  MoveL 8481 to (467.23, 529.71, 152) mm, rotated rx -180 ry 0 rz 160 deg; joints [10.696, 50.173, 8.575, -145.223, 63.505, 162.787]
  Set speed (16.9 mm/s)
  Call Extruder(111.55322)
  MoveL 8482 to (466.64, 529.05, 152) mm, rotated rx -180 ry 0 rz 160 deg; joints [10.622, 50.069, 8.779, -145.33, 63.566, 162.886]
  Set speed (16.9 mm/s)
  Call Extruder(114.56277)
  MoveL 8483 to (466.06, 528.36, 152) mm, rotated rx 180 ry 0 rz 160 deg; joints [10.545, 49.965, 8.983, -145.44, 63.625, 162.986]
  Call Extruder(117.70590)
  MoveL 8484 to (465.46, 527.63, 152) mm, rotated rx -180 ry 0 rz 160 deg; joints [10.463, 49.858, 9.191, -145.557, 63.685, 163.089]
  Set speed (16.9 mm/s)
  Call Extruder(120.63235)
  MoveL 8485 to (464.92, 526.94, 152) mm, rotated rx -180 ry 0 rz 160 deg; joints [10.384, 49.761, 9.381, -145.667, 63.739, 163.185]
  Call Extruder(123.51753)
  MoveL 8486 to (464.4, 526.25, 152) mm, rotated rx -180 ry 0 rz 160 deg; joints [10.304, 49.667, 9.565, -145.777, 63.79, 163.279]
  Set speed (16.9 mm/s)
  Call Extruder(126.65561)
  MoveL 8487 to (463.85, 525.49, 152) mm, rotated rx 180 ry 0 rz 160 deg; joints [10.215, 49.568, 9.76, -145.898, 63.844, 163.381]
  Set speed (16.9 mm/s)
  Call Extruder(130.52968)
  MoveL 8488 to (463.19, 524.53, 152) mm, rotated rx 180 ry 0 rz 160 deg; joints [10.102, 49.448, 9.995, -146.05, 63.907, 163.505]
  Call Extruder(135.63472)
  MoveL 8489 to (462.37, 523.24, 152) mm, rotated rx 180 ry 0 rz 160 deg; joints [9.948, 49.296, 10.292, -146.255, 63.984, 163.668]
  Set speed (16.9 mm/s)
  Call Extruder(138.64613)
  MoveL 8490 to (461.9, 522.47, 152) mm, rotated rx 180 ry 0 rz 160 deg; joints [9.855, 49.21, 10.461, -146.377, 64.027, 163.763]
  Set speed (16.9 mm/s)
  Call Extruder(141.85812)
  MoveL 8491 to (461.42, 521.64, 152) mm, rotated rx 180 ry 0 rz 160 deg; joints [9.753, 49.12, 10.637, -146.509, 64.07, 163.864]
  Set speed (16.9 mm/s)
  Call Extruder(144.69950)
  MoveL 8492 to (461.01, 520.89, 152) mm, rotated rx 180 ry 0 rz 160 deg; joints [9.661, 49.043, 10.788, -146.627, 64.107, 163.952]
  Set speed (16.9 mm/s)
  Call Extruder(147.76672)
  MoveL 8493 to (460.58, 520.07, 152) mm, rotated rx -180 ry 0 rz 160 deg; joints [9.56, 48.962, 10.946, -146.755, 64.144, 164.046]
  Set speed (16.9 mm/s)
  Call Extruder(150.71748)
  MoveL 8494 to (460.19, 519.28, 152) mm, rotated rx 180 ry 0 rz 160 deg; joints [9.461, 48.887, 11.094, -146.88, 64.177, 164.136]
  Call Extruder(156.72530)
  MoveL 8495 to (459.44, 517.64, 152) mm, rotated rx 180 ry 0 rz 160 deg; joints [9.255, 48.741, 11.38, -147.137, 64.239, 164.317]
  Call Extruder(162.74277)
  MoveL 8496 to (458.75, 515.98, 152) mm, rotated rx 180 ry 0 rz 160 deg; joints [9.042, 48.605, 11.647, -147.399, 64.292, 164.494]
  Set speed (16.9 mm/s)
  Call Extruder(164.64160)
  MoveL 8497 to (458.55, 515.44, 152) mm, rotated rx -180 ry 0 rz 160 deg; joints [8.974, 48.564, 11.727, -147.483, 64.306, 164.549]
  Set speed (16.9 mm/s)
  Call Extruder(168.87909)
  MoveL 8498 to (458.12, 514.25, 152) mm, rotated rx 180 ry 0 rz 160 deg; joints [8.819, 48.477, 11.898, -147.67, 64.336, 164.671]
  Set speed (16.9 mm/s)
  Call Extruder(174.83651)
  MoveL 8499 to (457.58, 512.55, 152) mm, rotated rx 180 ry 0 rz 160 deg; joints [8.596, 48.363, 12.122, -147.936, 64.37, 164.839]
  Call Extruder(180.93408)
  MoveL 8500 to (457.1, 510.79, 152) mm, rotated rx 180 ry 0 rz 160 deg; joints [8.363, 48.257, 12.33, -148.211, 64.396, 165.007]
  Set speed (16.9 mm/s)
  Call Extruder(186.95183)
  MoveL 8501 to (456.7, 509.03, 152) mm, rotated rx -180 ry 0 rz 160 deg; joints [8.128, 48.165, 12.512, -148.485, 64.412, 165.167]
  Set speed (16.9 mm/s)
  Call Extruder(193.18882)
  MoveL 8502 to (456.36, 507.19, 152) mm, rotated rx 180 ry 0 rz 160 deg; joints [7.881, 48.079, 12.679, -148.772, 64.419, 165.33]
  Set speed (16.9 mm/s)
  Call Extruder(199.22762)
  MoveL 8503 to (456.1, 505.4, 152) mm, rotated rx 180 ry 0 rz 160 deg; joints [7.637, 48.008, 12.818, -149.05, 64.416, 165.482]
  Set speed (16.9 mm/s)
  Call Extruder(205.26140)
  MoveL 8504 to (455.91, 503.6, 152) mm, rotated rx -180 ry 0 rz 160 deg; joints [7.39, 47.949, 12.936, -149.329, 64.404, 165.629]
  Set speed (16.9 mm/s)
  Call Extruder(211.19905)
  MoveL 8505 to (455.8, 501.82, 152) mm, rotated rx -180 ry 0 rz 160 deg; joints [7.145, 47.901, 13.029, -149.603, 64.382, 165.768]
  Set speed (16.9 mm/s)
  Call Extruder(217.23836)
  MoveL 8506 to (455.76, 500.01, 152) mm, rotated rx -180 ry 0 rz 160 deg; joints [6.894, 47.864, 13.102, -149.883, 64.352, 165.905]
  Set speed (16.9 mm/s)
  Call Extruder(222.75136)
  MoveL 8507 to (455.8, 498.36, 152) mm, rotated rx -180 ry 0 rz 160 deg; joints [6.662, 47.841, 13.147, -150.137, 64.315, 166.025]
  Set speed (16.9 mm/s)
  Call Extruder(228.09484)
  MoveL 8508 to (455.89, 496.76, 152) mm, rotated rx -180 ry 0 rz 160 deg; joints [6.438, 47.828, 13.173, -150.382, 64.272, 166.137]
  Call Extruder(233.51834)
  MoveL 8509 to (456.03, 495.14, 152) mm, rotated rx -180 ry 0 rz 160 deg; joints [6.209, 47.823, 13.182, -150.629, 64.222, 166.247]
  Call Extruder(238.82118)
  MoveL 8510 to (456.24, 493.56, 152) mm, rotated rx -180 ry 0 rz 160 deg; joints [5.986, 47.828, 13.172, -150.869, 64.164, 166.349]
  Set speed (16.9 mm/s)
  Call Extruder(244.49040)
  MoveL 8511 to (456.52, 491.89, 152) mm, rotated rx 180 ry 0 rz 160 deg; joints [5.748, 47.843, 13.142, -151.123, 64.096, 166.453]
  Call Extruder(249.82084)
  MoveL 8512 to (456.84, 490.32, 152) mm, rotated rx -180 ry 0 rz 160 deg; joints [5.525, 47.867, 13.096, -151.359, 64.024, 166.547]
  Set speed (16.9 mm/s)
  Call Extruder(255.25540)
  MoveL 8513 to (457.22, 488.74, 152) mm, rotated rx 180 ry 0 rz 160 deg; joints [5.298, 47.9, 13.03, -151.596, 63.943, 166.637]
  Set speed (16.9 mm/s)
  Call Extruder(260.70317)
  MoveL 8514 to (457.67, 487.17, 152) mm, rotated rx 180 ry 0 rz 160 deg; joints [5.073, 47.943, 12.946, -151.83, 63.855, 166.723]
  Set speed (16.9 mm/s)
  Call Extruder(266.12310)
  MoveL 8515 to (458.17, 485.63, 152) mm, rotated rx -180 ry 0 rz 160 deg; joints [4.851, 47.995, 12.844, -152.06, 63.76, 166.803]
  Set speed (16.9 mm/s)
  Call Extruder(271.65144)
  MoveL 8516 to (458.73, 484.07, 152) mm, rotated rx 180 ry 0 rz 160 deg; joints [4.628, 48.057, 12.722, -152.289, 63.656, 166.879]
  Call Extruder(277.08602)
  MoveL 8517 to (459.35, 482.56, 152) mm, rotated rx -180 ry 0 rz 160 deg; joints [4.411, 48.128, 12.584, -152.509, 63.546, 166.949]
  Call Extruder(282.51502)
  MoveL 8518 to (460.02, 481.08, 152) mm, rotated rx 180 ry 0 rz 160 deg; joints [4.197, 48.207, 12.428, -152.724, 63.43, 167.013]
  Call Extruder(287.86511)
  MoveL 8519 to (460.73, 479.64, 152) mm, rotated rx 180 ry 0 rz 160 deg; joints [3.99, 48.294, 12.257, -152.931, 63.309, 167.072]
  Set speed (16.9 mm/s)
  Call Extruder(293.30641)
  MoveL 8520 to (461.51, 478.21, 152) mm, rotated rx 180 ry 0 rz 160 deg; joints [3.783, 48.391, 12.066, -153.135, 63.18, 167.126]
  Set speed (16.9 mm/s)
  Call Extruder(298.82528)
  MoveL 8521 to (462.35, 476.78, 152) mm, rotated rx 180 ry 0 rz 160 deg; joints [3.578, 48.499, 11.854, -153.335, 63.041, 167.175]
  Set speed (16.9 mm/s)
  Call Extruder(304.15599)
  MoveL 8522 to (463.21, 475.44, 152) mm, rotated rx -180 ry 0 rz 160 deg; joints [3.385, 48.612, 11.634, -153.523, 62.902, 167.217]
  Set speed (16.9 mm/s)
  Call Extruder(309.59991)
  MoveL 8523 to (464.15, 474.1, 152) mm, rotated rx 180 ry 0 rz 160 deg; joints [3.192, 48.735, 11.392, -153.707, 62.753, 167.254]
  Set speed (16.9 mm/s)
  Call Extruder(315.02617)
  MoveL 8524 to (465.12, 472.8, 152) mm, rotated rx -180 ry 0 rz 160 deg; joints [3.005, 48.866, 11.136, -153.883, 62.599, 167.286]
  Set speed (16.9 mm/s)
  Call Extruder(320.54632)
  MoveL 8525 to (466.16, 471.51, 152) mm, rotated rx 180 ry 0 rz 160 deg; joints [2.821, 49.008, 10.858, -154.055, 62.436, 167.312]
  Set speed (16.9 mm/s)
  Call Extruder(325.88657)
  MoveL 8526 to (467.22, 470.31, 152) mm, rotated rx 180 ry 0 rz 160 deg; joints [2.648, 49.152, 10.574, -154.213, 62.273, 167.332]
  Call Extruder(331.41574)
  MoveL 8527 to (468.35, 469.1, 152) mm, rotated rx -180 ry 0 rz 160 deg; joints [2.476, 49.31, 10.265, -154.369, 62.099, 167.346]
  Set speed (16.9 mm/s)
  Call Extruder(336.75261)
  MoveL 8528 to (469.49, 467.97, 152) mm, rotated rx -180 ry 0 rz 160 deg; joints [2.315, 49.47, 9.952, -154.511, 61.926, 167.355]
  Set speed (16.9 mm/s)
  Call Extruder(342.18977)
  MoveL 8529 to (470.69, 466.87, 152) mm, rotated rx 180 ry 0 rz 160 deg; joints [2.159, 49.64, 9.619, -154.647, 61.744, 167.357]
  Call Extruder(347.70524)
  MoveL 8530 to (471.95, 465.8, 152) mm, rotated rx 180 ry 0 rz 160 deg; joints [2.006, 49.819, 9.268, -154.776, 61.555, 167.354]
  Set speed (16.9 mm/s)
  Call Extruder(353.50911)
  MoveL 8531 to (473.32, 464.72, 152) mm, rotated rx 180 ry 0 rz 160 deg; joints [1.854, 50.016, 8.883, -154.902, 61.352, 167.343]
  Set speed (16.9 mm/s)
  Call Extruder(357.99277)
  MoveL 8532 to (474.4, 463.93, 152) mm, rotated rx -180 ry 0 rz 160 deg; joints [1.742, 50.172, 8.576, -154.991, 61.191, 167.331]
  Set speed (16.9 mm/s)
  Call Extruder(363.92441)
  MoveL 8533 to (475.87, 462.93, 152) mm, rotated rx -180 ry 0 rz 160 deg; joints [1.602, 50.387, 8.156, -155.1, 60.974, 167.307]
  Set speed (16.9 mm/s)
  Call Extruder(369.45306)
  MoveL 8534 to (477.27, 462.05, 152) mm, rotated rx -180 ry 0 rz 160 deg; joints [1.479, 50.593, 7.752, -155.191, 60.768, 167.279]
  Set speed (16.9 mm/s)
  Call Extruder(374.88475)
  MoveL 8535 to (478.68, 461.24, 152) mm, rotated rx -180 ry 0 rz 160 deg; joints [1.365, 50.803, 7.343, -155.271, 60.561, 167.245]
  Call Extruder(380.22948)
  MoveL 8536 to (480.1, 460.5, 152) mm, rotated rx -180 ry 0 rz 160 deg; joints [1.261, 51.014, 6.93, -155.34, 60.355, 167.206]
  Call Extruder(385.74670)
  MoveL 8537 to (481.59, 459.78, 152) mm, rotated rx -180 ry 0 rz 160 deg; joints [1.162, 51.237, 6.493, -155.401, 60.138, 167.159]
  Set speed (16.9 mm/s)
  Call Extruder(391.17918)
  MoveL 8538 to (483.09, 459.13, 152) mm, rotated rx 180 ry 0 rz 160 deg; joints [1.072, 51.463, 6.052, -155.451, 59.922, 167.106]
  Call Extruder(396.52455)
  MoveL 8539 to (484.58, 458.54, 152) mm, rotated rx -180 ry 0 rz 160 deg; joints [0.99, 51.689, 5.609, -155.49, 59.708, 167.048]
  Set speed (16.9 mm/s)
  Call Extruder(402.01351)
  MoveL 8540 to (486.13, 458, 152) mm, rotated rx 180 ry 0 rz 160 deg; joints [0.915, 51.926, 5.146, -155.52, 59.485, 166.982]
  Call Extruder(407.42300)
  MoveL 8541 to (487.68, 457.52, 152) mm, rotated rx 180 ry 0 rz 160 deg; joints [0.849, 52.164, 4.681, -155.539, 59.264, 166.911]
  Set speed (16.9 mm/s)
  Call Extruder(412.57446)
  MoveL 8542 to (489.17, 457.11, 152) mm, rotated rx -180 ry 0 rz 160 deg; joints [0.793, 52.395, 4.231, -155.548, 59.051, 166.838]
  Set speed (16.9 mm/s)
  Call Extruder(418.05427)
  MoveL 8543 to (490.77, 456.74, 152) mm, rotated rx 180 ry 0 rz 160 deg; joints [0.742, 52.643, 3.746, -155.547, 58.824, 166.754]
  Call Extruder(423.53685)
  MoveL 8544 to (492.38, 456.43, 152) mm, rotated rx -180 ry 0 rz 160 deg; joints [0.699, 52.896, 3.253, -155.536, 58.595, 166.663]
  Set speed (16.9 mm/s)
  Call Extruder(429.18834)
  MoveL 8545 to (494.06, 456.17, 152) mm, rotated rx 180 ry 0 rz 160 deg; joints [0.662, 53.159, 2.739, -155.514, 58.359, 166.563]
  Set speed (16.9 mm/s)
  Call Extruder(434.59269)
  MoveL 8546 to (495.66, 455.98, 152) mm, rotated rx -180 ry 0 rz 160 deg; joints [0.636, 53.414, 2.242, -155.482, 58.132, 166.461]
  Set speed (16.9 mm/s)
  Call Extruder(440.01240)
  MoveL 8547 to (497.28, 455.85, 152) mm, rotated rx 180 ry 0 rz 160 deg; joints [0.617, 53.672, 1.739, -155.44, 57.905, 166.352]
  Set speed (16.9 mm/s)
  Call Extruder(445.51598)
  MoveL 8548 to (498.93, 455.78, 152) mm, rotated rx -180 ry 0 rz 160 deg; joints [0.606, 53.936, 1.224, -155.388, 57.674, 166.236]
  Set speed (16.9 mm/s)
  Call Extruder(450.85230)
  MoveL 8549 to (500.53, 455.77, 152) mm, rotated rx 180 ry 0 rz 160 deg; joints [0.602, 54.194, 0.722, -155.327, 57.451, 166.117]
  Set speed (16.9 mm/s)
  Call Extruder(456.35038)
  MoveL 8550 to (502.18, 455.82, 152) mm, rotated rx -180 ry 0 rz 160 deg; joints [0.606, 54.462, 0.2, -155.254, 57.222, 165.988]
  Set speed (16.9 mm/s)
  Call Extruder(461.73242)
  MoveL 8551 to (503.79, 455.93, 152) mm, rotated rx -180 ry 0 rz 160 deg; joints [0.618, 54.725, -0.312, -155.173, 56.998, 165.857]
  Set speed (16.9 mm/s)
  Call Extruder(467.24230)
  MoveL 8552 to (505.43, 456.1, 152) mm, rotated rx 180 ry 0 rz 160 deg; joints [0.637, 54.995, -0.838, -155.08, 56.771, 165.716]
  Set speed (16.9 mm/s)
  Call Extruder(472.59761)
  MoveL 8553 to (507.02, 456.33, 152) mm, rotated rx 180 ry 0 rz 160 deg; joints [0.664, 55.258, -1.349, -154.981, 56.552, 165.574]
  Call Extruder(478.00070)
  MoveL 8554 to (508.62, 456.61, 152) mm, rotated rx 180 ry 0 rz 160 deg; joints [0.697, 55.523, -1.866, -154.871, 56.333, 165.424]
  Set speed (16.9 mm/s)
  Call Extruder(482.76006)
  MoveL 8555 to (510.01, 456.91, 152) mm, rotated rx -180 ry 0 rz 160 deg; joints [0.732, 55.757, -2.32, -154.767, 56.142, 165.289]
  Call Extruder(488.88102)
  MoveL 8556 to (511.79, 457.37, 152) mm, rotated rx -180 ry 0 rz 160 deg; joints [0.786, 56.057, -2.904, -154.624, 55.899, 165.108]
  Set speed (16.9 mm/s)
  Call Extruder(494.30171)
  MoveL 8557 to (513.34, 457.83, 152) mm, rotated rx 180 ry 0 rz 160 deg; joints [0.84, 56.322, -3.419, -154.487, 55.687, 164.942]
  Call Extruder(499.82708)
  MoveL 8558 to (514.91, 458.36, 152) mm, rotated rx 180 ry 0 rz 160 deg; joints [0.903, 56.59, -3.942, -154.339, 55.475, 164.768]
  Call Extruder(505.16704)
  MoveL 8559 to (516.41, 458.93, 152) mm, rotated rx 180 ry 0 rz 160 deg; joints [0.97, 56.849, -4.444, -154.187, 55.273, 164.595]
  Set speed (16.9 mm/s)
  Call Extruder(510.69488)
  MoveL 8560 to (517.94, 459.57, 152) mm, rotated rx -180 ry 0 rz 160 deg; joints [1.045, 57.114, -4.96, -154.022, 55.068, 164.411]
  Set speed (16.9 mm/s)
  Call Extruder(516.02911)
  MoveL 8561 to (519.39, 460.24, 152) mm, rotated rx -180 ry 0 rz 160 deg; joints [1.125, 57.368, -5.453, -153.855, 54.874, 164.229]
  Set speed (16.9 mm/s)
  Call Extruder(521.56196)
  MoveL 8562 to (520.87, 461, 152) mm, rotated rx 180 ry 0 rz 160 deg; joints [1.213, 57.629, -5.959, -153.674, 54.678, 164.036]
  Set speed (16.9 mm/s)
  Call Extruder(526.98931)
  MoveL 8563 to (522.28, 461.79, 152) mm, rotated rx 180 ry 0 rz 160 deg; joints [1.306, 57.882, -6.45, -153.49, 54.491, 163.842]
  Set speed (16.9 mm/s)
  Call Extruder(532.32683)
  MoveL 8564 to (523.65, 462.62, 152) mm, rotated rx 180 ry 0 rz 160 deg; joints [1.403, 58.127, -6.926, -153.301, 54.311, 163.649]
  Set speed (16.9 mm/s)
  Call Extruder(537.85094)
  MoveL 8565 to (525.03, 463.53, 152) mm, rotated rx -180 ry 0 rz 160 deg; joints [1.509, 58.378, -7.412, -153.1, 54.131, 163.445]
  Set speed (16.9 mm/s)
  Call Extruder(543.19366)
  MoveL 8566 to (526.34, 464.46, 152) mm, rotated rx -180 ry 0 rz 160 deg; joints [1.616, 58.616, -7.874, -152.898, 53.963, 163.244]
  Set speed (16.9 mm/s)
  Call Extruder(548.66042)
  MoveL 8567 to (527.64, 465.47, 152) mm, rotated rx 180 ry 0 rz 160 deg; joints [1.732, 58.855, -8.338, -152.686, 53.796, 163.036]
  Call Extruder(554.09541)
  MoveL 8568 to (528.89, 466.51, 152) mm, rotated rx 180 ry 0 rz 160 deg; joints [1.852, 59.088, -8.79, -152.47, 53.637, 162.827]
  Set speed (16.9 mm/s)
  Call Extruder(559.59156)
  MoveL 8569 to (530.12, 467.61, 152) mm, rotated rx -180 ry 0 rz 160 deg; joints [1.979, 59.319, -9.237, -152.246, 53.483, 162.613]
  Call Extruder(564.97166)
  MoveL 8570 to (531.28, 468.73, 152) mm, rotated rx 180 ry 0 rz 160 deg; joints [2.107, 59.539, -9.664, -152.021, 53.339, 162.401]
  Set speed (16.9 mm/s)
  Call Extruder(567.88723)
  MoveL 8571 to (531.89, 469.35, 152) mm, rotated rx -180 ry 0 rz 160 deg; joints [2.179, 59.656, -9.891, -151.898, 53.264, 162.286]
  Call Extruder(570.83929)
  MoveL 8572 to (532.5, 469.99, 152) mm, rotated rx 180 ry 0 rz 160 deg; joints [2.253, 59.773, -10.117, -151.771, 53.19, 162.169]
  Set speed (16.9 mm/s)
  Call Extruder(573.85291)
  MoveL 8573 to (533.11, 470.66, 152) mm, rotated rx -180 ry 0 rz 160 deg; joints [2.329, 59.891, -10.345, -151.641, 53.116, 162.049]
  Set speed (16.9 mm/s)
  Call Extruder(576.90040)
  MoveL 8574 to (533.7, 471.35, 152) mm, rotated rx -180 ry 0 rz 160 deg; joints [2.408, 60.007, -10.571, -151.508, 53.045, 161.928]
  Set speed (16.9 mm/s)
  Call Extruder(579.88352)
  MoveL 8575 to (534.27, 472.04, 152) mm, rotated rx 180 ry 0 rz 160 deg; joints [2.486, 60.119, -10.788, -151.377, 52.977, 161.809]
  Set speed (16.9 mm/s)
  Call Extruder(582.95706)
  MoveL 8576 to (534.85, 472.76, 152) mm, rotated rx 180 ry 0 rz 160 deg; joints [2.569, 60.233, -11.008, -151.241, 52.909, 161.686]
  Set speed (16.9 mm/s)
  Call Extruder(585.93160)
  MoveL 8577 to (535.39, 473.47, 152) mm, rotated rx 180 ry 0 rz 160 deg; joints [2.649, 60.341, -11.217, -151.108, 52.846, 161.567]
  Set speed (16.9 mm/s)
  Call Extruder(589.06730)
  MoveL 8578 to (535.95, 474.23, 152) mm, rotated rx -180 ry 0 rz 160 deg; joints [2.735, 60.452, -11.432, -150.967, 52.782, 161.442]
  Set speed (16.9 mm/s)
  Call Extruder(591.96265)
  MoveL 8579 to (536.45, 474.94, 152) mm, rotated rx -180 ry 0 rz 160 deg; joints [2.816, 60.553, -11.627, -150.836, 52.726, 161.326]
  Set speed (16.9 mm/s)
  Call Extruder(594.99815)
  MoveL 8580 to (536.95, 475.69, 152) mm, rotated rx 180 ry 0 rz 160 deg; joints [2.902, 60.656, -11.827, -150.698, 52.669, 161.205]
  Call Extruder(598.05624)
  MoveL 8581 to (537.45, 476.46, 152) mm, rotated rx -180 ry 0 rz 160 deg; joints [2.99, 60.758, -12.024, -150.558, 52.614, 161.083]
  Call Extruder(601.06718)
  MoveL 8582 to (537.92, 477.23, 152) mm, rotated rx -180 ry 0 rz 160 deg; joints [3.077, 60.855, -12.212, -150.42, 52.564, 160.963]
  Set speed (16.9 mm/s)
  Call Extruder(604.06606)
  MoveL 8583 to (538.38, 478.01, 152) mm, rotated rx -180 ry 0 rz 160 deg; joints [3.165, 60.95, -12.397, -150.281, 52.515, 160.844]
  Set speed (16.9 mm/s)
  Call Extruder(608.88178)
  MoveL 8584 to (539.08, 479.27, 152) mm, rotated rx 180 ry 0 rz 160 deg; joints [3.308, 61.098, -12.682, -150.059, 52.442, 160.654]
  Call Extruder(613.09280)
  MoveL 8585 to (539.65, 480.39, 152) mm, rotated rx 180 ry 0 rz 160 deg; joints [3.435, 61.22, -12.92, -149.863, 52.385, 160.489]
  Set speed (16.9 mm/s)
  Call Extruder(616.12747)
  MoveL 8586 to (540.04, 481.21, 152) mm, rotated rx 180 ry 0 rz 160 deg; joints [3.528, 61.306, -13.085, -149.721, 52.347, 160.371]
  Set speed (16.9 mm/s)
  Call Extruder(619.14351)
  MoveL 8587 to (540.42, 482.03, 152) mm, rotated rx 180 ry 0 rz 160 deg; joints [3.621, 61.389, -13.245, -149.58, 52.312, 160.254]
  Set speed (16.9 mm/s)
  Call Extruder(625.34531)
  MoveL 8588 to (541.14, 483.75, 152) mm, rotated rx 180 ry 0 rz 160 deg; joints [3.815, 61.549, -13.555, -149.291, 52.249, 160.016]
  Set speed (16.9 mm/s)
  Call Extruder(631.18422)
  MoveL 8589 to (541.75, 485.39, 152) mm, rotated rx -180 ry 0 rz 160 deg; joints [4.001, 61.689, -13.827, -149.018, 52.2, 159.796]
  Set speed (16.9 mm/s)
  Call Extruder(637.24238)
  MoveL 8590 to (542.31, 487.11, 152) mm, rotated rx 180 ry 0 rz 160 deg; joints [4.196, 61.824, -14.087, -148.735, 52.16, 159.571]
  Set speed (16.9 mm/s)
  Call Extruder(643.43589)
  MoveL 8591 to (542.82, 488.9, 152) mm, rotated rx 180 ry 0 rz 160 deg; joints [4.399, 61.949, -14.329, -148.448, 52.132, 159.347]
  Set speed (16.9 mm/s)
  Call Extruder(649.40759)
  MoveL 8592 to (543.23, 490.64, 152) mm, rotated rx 180 ry 0 rz 160 deg; joints [4.597, 62.057, -14.538, -148.172, 52.116, 159.136]
  Set speed (16.9 mm/s)
  Call Extruder(655.48431)
  MoveL 8593 to (543.58, 492.43, 152) mm, rotated rx 180 ry 0 rz 160 deg; joints [4.8, 62.155, -14.726, -147.894, 52.112, 158.927]
  Set speed (16.9 mm/s)
  Call Extruder(661.50732)
  MoveL 8594 to (543.85, 494.21, 152) mm, rotated rx 180 ry 0 rz 160 deg; joints [5.003, 62.239, -14.889, -147.622, 52.119, 158.727]
  Call Extruder(667.39278)
  MoveL 8595 to (544.05, 495.96, 152) mm, rotated rx -180 ry 0 rz 160 deg; joints [5.203, 62.308, -15.023, -147.359, 52.137, 158.538]
  Set speed (16.9 mm/s)
  Call Extruder(673.59529)
  MoveL 8596 to (544.18, 497.82, 152) mm, rotated rx -180 ry 0 rz 160 deg; joints [5.415, 62.369, -15.14, -147.085, 52.167, 158.346]
  Set speed (16.9 mm/s)
  Call Extruder(679.61986)
  MoveL 8597 to (544.23, 499.63, 152) mm, rotated rx 180 ry 0 rz 160 deg; joints [5.622, 62.414, -15.227, -146.824, 52.209, 158.168]
  Call Extruder(685.75246)
  MoveL 8598 to (544.21, 501.46, 152) mm, rotated rx 180 ry 0 rz 160 deg; joints [5.834, 62.446, -15.289, -146.563, 52.263, 157.995]
  Call Extruder(691.68280)
  MoveL 8599 to (544.12, 503.24, 152) mm, rotated rx 180 ry 0 rz 160 deg; joints [6.039, 62.464, -15.324, -146.315, 52.326, 157.836]
  Set speed (16.9 mm/s)
  Call Extruder(697.71345)
  MoveL 8600 to (543.95, 505.04, 152) mm, rotated rx 180 ry 0 rz 160 deg; joints [6.248, 62.469, -15.334, -146.069, 52.401, 157.684]
  Set speed (16.9 mm/s)
  Call Extruder(703.84606)
  MoveL 8601 to (543.7, 506.86, 152) mm, rotated rx 180 ry 0 rz 160 deg; joints [6.46, 62.46, -15.316, -145.825, 52.489, 157.539]
  Set speed (16.9 mm/s)
  Call Extruder(709.77348)
  MoveL 8602 to (543.39, 508.61, 152) mm, rotated rx -180 ry 0 rz 160 deg; joints [6.665, 62.438, -15.274, -145.596, 52.585, 157.408]
  Call Extruder(715.61424)
  MoveL 8603 to (543.01, 510.32, 152) mm, rotated rx 180 ry 0 rz 160 deg; joints [6.866, 62.404, -15.208, -145.376, 52.688, 157.289]
  Set speed (16.9 mm/s)
  Call Extruder(721.80459)
  MoveL 8604 to (542.54, 512.12, 152) mm, rotated rx -180 ry 0 rz 160 deg; joints [7.079, 62.354, -15.112, -145.15, 52.809, 157.173]
  Set speed (16.9 mm/s)
  Call Extruder(727.90138)
  MoveL 8605 to (542, 513.87, 152) mm, rotated rx 180 ry 0 rz 160 deg; joints [7.287, 62.292, -14.991, -144.934, 52.937, 157.07]
  Call Extruder(734.04898)
  MoveL 8606 to (541.39, 515.6, 152) mm, rotated rx 180 ry 0 rz 160 deg; joints [7.496, 62.216, -14.844, -144.725, 53.077, 156.976]
  Set speed (16.9 mm/s)
  Call Extruder(739.76790)
  MoveL 8607 to (540.75, 517.2, 152) mm, rotated rx 180 ry 0 rz 160 deg; joints [7.688, 62.132, -14.683, -144.537, 53.216, 156.9]
  Set speed (16.9 mm/s)
  Call Extruder(745.87332)
  MoveL 8608 to (540.01, 518.87, 152) mm, rotated rx 180 ry 0 rz 160 deg; joints [7.892, 62.031, -14.487, -144.345, 53.373, 156.829]
  Set speed (16.9 mm/s)
  Call Extruder(748.95640)
  MoveL 8609 to (539.61, 519.7, 152) mm, rotated rx 180 ry 0 rz 160 deg; joints [7.994, 61.975, -14.379, -144.251, 53.455, 156.797]
  Set speed (16.9 mm/s)
  Call Extruder(751.90685)
  MoveL 8610 to (539.2, 520.49, 152) mm, rotated rx -180 ry 0 rz 160 deg; joints [8.091, 61.918, -14.269, -144.162, 53.536, 156.77]
  Set speed (16.9 mm/s)
  Call Extruder(755.31926)
  MoveL 8611 to (538.72, 521.39, 152) mm, rotated rx 180 ry 0 rz 160 deg; joints [8.203, 61.85, -14.136, -144.063, 53.632, 156.741]
  Set speed (16.9 mm/s)
  Call Extruder(758.08631)
  MoveL 8612 to (538.31, 522.11, 152) mm, rotated rx 180 ry 0 rz 160 deg; joints [8.292, 61.79, -14.021, -143.984, 53.713, 156.721]
  Set speed (16.9 mm/s)
  Call Extruder(763.51652)
  MoveL 8613 to (537.48, 523.5, 152) mm, rotated rx 180 ry 0 rz 160 deg; joints [8.467, 61.668, -13.786, -143.834, 53.874, 156.686]
  Set speed (16.9 mm/s)
  Call Extruder(766.36303)
  MoveL 8614 to (537.01, 524.22, 152) mm, rotated rx 180 ry 0 rz 160 deg; joints [8.558, 61.6, -13.653, -143.759, 53.961, 156.672]
  Set speed (16.9 mm/s)
  Call Extruder(771.70559)
  MoveL 8615 to (536.11, 525.55, 152) mm, rotated rx 180 ry 0 rz 160 deg; joints [8.726, 61.466, -13.394, -143.621, 54.129, 156.651]
  Set speed (16.9 mm/s)
  Call Extruder(776.09850)
  MoveL 8616 to (535.33, 526.61, 152) mm, rotated rx 180 ry 0 rz 160 deg; joints [8.863, 61.348, -13.166, -143.514, 54.272, 156.642]
  Set speed (16.9 mm/s)
  Call Extruder(779.07385)
  MoveL 8617 to (534.79, 527.32, 152) mm, rotated rx 180 ry 0 rz 160 deg; joints [8.954, 61.265, -13.007, -143.444, 54.37, 156.638]
  Set speed (16.9 mm/s)
  Call Extruder(782.31334)
  MoveL 8618 to (534.18, 528.07, 152) mm, rotated rx 180 ry 0 rz 160 deg; joints [9.053, 61.172, -12.826, -143.369, 54.479, 156.637]
  Set speed (16.9 mm/s)
  Call Extruder(785.08810)
  MoveL 8619 to (533.65, 528.71, 152) mm, rotated rx 180 ry 0 rz 160 deg; joints [9.136, 61.09, -12.668, -143.308, 54.574, 156.639]
  Set speed (16.9 mm/s)
  Call Extruder(788.18970)
  MoveL 8620 to (533.04, 529.41, 152) mm, rotated rx 180 ry 0 rz 160 deg; joints [9.229, 60.996, -12.485, -143.241, 54.681, 156.643]
  Call Extruder(791.17742)
  MoveL 8621 to (532.44, 530.08, 152) mm, rotated rx 180 ry 0 rz 160 deg; joints [9.317, 60.903, -12.305, -143.179, 54.785, 156.649]
  Call Extruder(794.30638)
  MoveL 8622 to (531.79, 530.76, 152) mm, rotated rx 180 ry 0 rz 160 deg; joints [9.409, 60.803, -12.112, -143.116, 54.897, 156.659]
  Set speed (16.9 mm/s)
  Call Extruder(797.24483)
  MoveL 8623 to (531.17, 531.38, 152) mm, rotated rx -180 ry 0 rz 160 deg; joints [9.493, 60.706, -11.924, -143.059, 55.002, 156.671]
  Set speed (16.9 mm/s)
  Call Extruder(800.21250)
  MoveL 8624 to (530.53, 532, 152) mm, rotated rx -180 ry 0 rz 160 deg; joints [9.578, 60.606, -11.731, -143.004, 55.111, 156.685]
  Call Extruder(803.23832)
  MoveL 8625 to (529.87, 532.62, 152) mm, rotated rx 180 ry 0 rz 160 deg; joints [9.663, 60.502, -11.529, -142.949, 55.222, 156.703]
  Set speed (16.9 mm/s)
  Call Extruder(806.30324)
  MoveL 8626 to (529.19, 533.24, 152) mm, rotated rx -180 ry 0 rz 160 deg; joints [9.748, 60.394, -11.321, -142.897, 55.336, 156.722]
  Set speed (16.9 mm/s)
  Call Extruder(809.25471)
  MoveL 8627 to (528.51, 533.82, 152) mm, rotated rx -180 ry 0 rz 160 deg; joints [9.828, 60.288, -11.115, -142.848, 55.447, 156.744]
  Set speed (16.9 mm/s)
  Call Extruder(812.46812)
  MoveL 8628 to (527.77, 534.43, 152) mm, rotated rx -180 ry 0 rz 160 deg; joints [9.915, 60.171, -10.888, -142.797, 55.569, 156.77]
  Set speed (16.9 mm/s)
  Call Extruder(815.31986)
  MoveL 8629 to (527.1, 534.96, 152) mm, rotated rx 180 ry 0 rz 160 deg; joints [9.99, 60.064, -10.682, -142.754, 55.678, 156.796]
  Set speed (16.9 mm/s)
  Call Extruder(818.31128)
  MoveL 8630 to (526.39, 535.5, 152) mm, rotated rx 180 ry 0 rz 160 deg; joints [10.068, 59.951, -10.461, -142.712, 55.794, 156.825]
  Call Extruder(821.38972)
  MoveL 8631 to (525.64, 536.04, 152) mm, rotated rx 180 ry 0 rz 160 deg; joints [10.147, 59.832, -10.231, -142.67, 55.913, 156.857]
  Call Extruder(824.35422)
  MoveL 8632 to (524.91, 536.55, 152) mm, rotated rx 180 ry 0 rz 160 deg; joints [10.222, 59.715, -10.006, -142.631, 56.029, 156.891]
  Set speed (16.9 mm/s)
  Call Extruder(827.52385)
  MoveL 8633 to (524.12, 537.08, 152) mm, rotated rx -180 ry 0 rz 160 deg; joints [10.301, 59.589, -9.761, -142.593, 56.154, 156.929]
  Set speed (16.9 mm/s)
  Call Extruder(830.38922)
  MoveL 8634 to (523.4, 537.54, 152) mm, rotated rx 180 ry 0 rz 160 deg; joints [10.37, 59.473, -9.536, -142.56, 56.268, 156.966]
  Call Extruder(833.47044)
  MoveL 8635 to (522.61, 538.02, 152) mm, rotated rx 180 ry 0 rz 160 deg; joints [10.443, 59.346, -9.291, -142.527, 56.391, 157.008]
  Set speed (16.9 mm/s)
  Call Extruder(836.39963)
  MoveL 8636 to (521.85, 538.46, 152) mm, rotated rx 180 ry 0 rz 160 deg; joints [10.512, 59.225, -9.055, -142.497, 56.508, 157.049]
  Set speed (16.9 mm/s)
  Call Extruder(838.90846)
  MoveL 8637 to (521.19, 538.83, 152) mm, rotated rx -180 ry 0 rz 160 deg; joints [10.569, 59.119, -8.851, -142.474, 56.609, 157.086]
  Set speed (16.9 mm/s)
  Call Extruder(844.21471)
  MoveL 8638 to (519.78, 539.57, 152) mm, rotated rx 180 ry 0 rz 160 deg; joints [10.687, 58.893, -8.412, -142.429, 56.823, 157.17]
  Set speed (16.9 mm/s)
  Call Extruder(848.68539)
  MoveL 8639 to (518.58, 540.14, 152) mm, rotated rx -180 ry 0 rz 160 deg; joints [10.782, 58.698, -8.034, -142.397, 57.005, 157.246]
  Set speed (16.9 mm/s)
  Call Extruder(854.58758)
  MoveL 8640 to (516.96, 540.86, 152) mm, rotated rx 180 ry 0 rz 160 deg; joints [10.904, 58.437, -7.527, -142.361, 57.247, 157.352]
  Set speed (16.9 mm/s)
  Call Extruder(860.52564)
  MoveL 8641 to (515.3, 541.5, 152) mm, rotated rx -180 ry 0 rz 160 deg; joints [11.019, 58.168, -7.006, -142.333, 57.491, 157.467]
  Set speed (16.9 mm/s)
  Call Extruder(866.62818)
  MoveL 8642 to (513.57, 542.1, 152) mm, rotated rx 180 ry 0 rz 160 deg; joints [11.13, 57.888, -6.462, -142.314, 57.742, 157.593]
  Set speed (16.9 mm/s)
  Call Extruder(872.53568)
  MoveL 8643 to (511.87, 542.61, 152) mm, rotated rx -180 ry 0 rz 160 deg; joints [11.231, 57.613, -5.928, -142.303, 57.985, 157.721]
  Set speed (16.9 mm/s)
  Call Extruder(875.22946)
  MoveL 8644 to (511.1, 542.82, 152) mm, rotated rx -180 ry 0 rz 160 deg; joints [11.274, 57.486, -5.681, -142.301, 58.096, 157.783]
  Set speed (16.9 mm/s)
  Call Extruder(878.68714)
  MoveL 8645 to (510.09, 543.07, 152) mm, rotated rx 180 ry 0 rz 160 deg; joints [11.328, 57.323, -5.364, -142.301, 58.238, 157.862]
  Set speed (16.9 mm/s)
  Call Extruder(884.86642)
  MoveL 8646 to (508.28, 543.45, 152) mm, rotated rx 180 ry 0 rz 160 deg; joints [11.418, 57.028, -4.791, -142.308, 58.492, 158.011]
  Call Extruder(890.96292)
  MoveL 8647 to (506.48, 543.76, 152) mm, rotated rx -180 ry 0 rz 160 deg; joints [11.499, 56.734, -4.221, -142.323, 58.741, 158.163]
  Call Extruder(896.90187)
  MoveL 8648 to (504.71, 543.98, 152) mm, rotated rx -180 ry 0 rz 160 deg; joints [11.57, 56.446, -3.661, -142.347, 58.983, 158.317]
  Call Extruder(902.97856)
  MoveL 8649 to (502.89, 544.14, 152) mm, rotated rx 180 ry 0 rz 160 deg; joints [11.634, 56.149, -3.084, -142.38, 59.228, 158.481]
  Set speed (16.9 mm/s)
  Call Extruder(909.08690)
  MoveL 8650 to (501.07, 544.22, 152) mm, rotated rx 180 ry 0 rz 160 deg; joints [11.69, 55.85, -2.503, -142.421, 59.472, 158.651]
  Set speed (16.9 mm/s)
  Call Extruder(915.02014)
  MoveL 8651 to (499.29, 544.23, 152) mm, rotated rx -180 ry 0 rz 160 deg; joints [11.736, 55.559, -1.936, -142.47, 59.707, 158.82]
  Set speed (10.0 mm/s)
  MoveL 8652 to (499.29, 544.23, 156) mm, rotated rx 180 ry 0 rz 160 deg; joints [11.736, 54.99, -1.803, -142.313, 59.362, 158.511]
  Set speed (120.0 mm/s)
  MoveL 8653 to (499.34, 542.82, 156) mm, rotated rx 180 ry 0 rz 160 deg; joints [11.562, 54.951, -1.727, -142.515, 59.328, 158.634]
  Set speed (17.0 mm/s)
  Call Extruder(920.96697)
  MoveL 8654 to (497.54, 542.75, 156) mm, rotated rx 180 ry 0 rz 160 deg; joints [11.599, 54.655, -1.154, -142.574, 59.56, 158.808]
  Set speed (17.0 mm/s)
  Call Extruder(926.80341)
  MoveL 8655 to (495.79, 542.62, 156) mm, rotated rx 180 ry 0 rz 160 deg; joints [11.626, 54.364, -0.593, -142.641, 59.786, 158.984]
  Call Extruder(932.71068)
  MoveL 8656 to (494.02, 542.4, 156) mm, rotated rx 180 ry 0 rz 160 deg; joints [11.645, 54.071, -0.026, -142.717, 60.01, 159.166]
  Call Extruder(938.64226)
  MoveL 8657 to (492.25, 542.12, 156) mm, rotated rx -180 ry 0 rz 160 deg; joints [11.655, 53.778, 0.541, -142.801, 60.232, 159.352]
  Set speed (17.0 mm/s)
  Call Extruder(944.27319)
  MoveL 8658 to (490.58, 541.78, 156) mm, rotated rx 180 ry 0 rz 160 deg; joints [11.655, 53.501, 1.077, -142.89, 60.438, 159.531]
  Set speed (17.0 mm/s)
  Call Extruder(950.10735)
  MoveL 8659 to (488.87, 541.35, 156) mm, rotated rx 180 ry 0 rz 160 deg; joints [11.646, 53.216, 1.628, -142.99, 60.648, 159.72]
  Set speed (17.0 mm/s)
  Call Extruder(955.69601)
  MoveL 8660 to (487.25, 540.88, 156) mm, rotated rx 180 ry 0 rz 160 deg; joints [11.629, 52.946, 2.152, -143.094, 60.844, 159.904]
  Call Extruder(961.71829)
  MoveL 8661 to (485.53, 540.3, 156) mm, rotated rx 180 ry 0 rz 160 deg; joints [11.601, 52.657, 2.711, -143.214, 61.051, 160.104]
  Set speed (17.0 mm/s)
  Call Extruder(967.31698)
  MoveL 8662 to (483.95, 539.7, 156) mm, rotated rx -180 ry 0 rz 160 deg; joints [11.566, 52.392, 3.225, -143.334, 61.238, 160.292]
  Set speed (17.0 mm/s)
  Call Extruder(972.99448)
  MoveL 8663 to (482.38, 539.03, 156) mm, rotated rx 180 ry 0 rz 160 deg; joints [11.521, 52.126, 3.739, -143.464, 61.423, 160.484]
  Set speed (17.0 mm/s)
  Call Extruder(976.15918)
  MoveL 8664 to (481.51, 538.63, 156) mm, rotated rx -180 ry 0 rz 160 deg; joints [11.492, 51.98, 4.023, -143.539, 61.524, 160.592]
  Set speed (17.0 mm/s)
  Call Extruder(980.07387)
  MoveL 8665 to (480.45, 538.1, 156) mm, rotated rx -180 ry 0 rz 160 deg; joints [11.453, 51.801, 4.37, -143.635, 61.646, 160.725]
  Set speed (17.0 mm/s)
  Call Extruder(984.71518)
  MoveL 8666 to (479.22, 537.44, 156) mm, rotated rx -180 ry 0 rz 160 deg; joints [11.4, 51.591, 4.776, -143.754, 61.787, 160.884]
  Set speed (17.0 mm/s)
  Call Extruder(987.60539)
  MoveL 8667 to (478.46, 537.01, 156) mm, rotated rx -180 ry 0 rz 160 deg; joints [11.364, 51.462, 5.026, -143.831, 61.873, 160.984]
  Set speed (17.0 mm/s)
  Call Extruder(991.38181)
  MoveL 8668 to (477.48, 536.43, 156) mm, rotated rx -180 ry 0 rz 160 deg; joints [11.314, 51.295, 5.35, -143.934, 61.983, 161.114]
  Set speed (17.0 mm/s)
  Call Extruder(995.83211)
  MoveL 8669 to (476.35, 535.7, 156) mm, rotated rx 180 ry 0 rz 160 deg; joints [11.25, 51.101, 5.726, -144.06, 62.109, 161.267]
  Set speed (17.0 mm/s)
  Call Extruder(999.28816)
  MoveL 8670 to (475.49, 535.11, 156) mm, rotated rx 180 ry 0 rz 160 deg; joints [11.195, 50.953, 6.012, -144.161, 62.204, 161.386]
  Set speed (17.0 mm/s)
  Call Extruder(1002.10754)
  MoveL 8671 to (474.79, 534.62, 156) mm, rotated rx -180 ry 0 rz 160 deg; joints [11.149, 50.834, 6.244, -144.245, 62.281, 161.483]
  Set speed (17.1 mm/s)
  Call Extruder(1005.56985)
  MoveL 8672 to (473.96, 533.99, 156) mm, rotated rx 180 ry 0 rz 160 deg; joints [11.089, 50.689, 6.525, -144.351, 62.372, 161.603]
  Set speed (17.0 mm/s)
  Call Extruder(1010.78368)
  MoveL 8673 to (472.72, 533.01, 156) mm, rotated rx 180 ry 0 rz 160 deg; joints [10.992, 50.476, 6.939, -144.515, 62.505, 161.782]
  Set speed (17.0 mm/s)
  Call Extruder(1013.88004)
  MoveL 8674 to (472.01, 532.41, 156) mm, rotated rx 180 ry 0 rz 160 deg; joints [10.931, 50.351, 7.18, -144.616, 62.581, 161.889]
  Call Extruder(1016.65899)
  MoveL 8675 to (471.38, 531.85, 156) mm, rotated rx -180 ry 0 rz 160 deg; joints [10.874, 50.242, 7.393, -144.708, 62.648, 161.984]
  Set speed (17.0 mm/s)
  Call Extruder(1021.02071)
  MoveL 8676 to (470.41, 530.96, 156) mm, rotated rx -180 ry 0 rz 160 deg; joints [10.781, 50.072, 7.722, -144.855, 62.749, 162.133]
  Call Extruder(1025.35782)
  MoveL 8677 to (469.48, 530.04, 156) mm, rotated rx 180 ry 0 rz 160 deg; joints [10.683, 49.908, 8.041, -145.005, 62.846, 162.281]
  Set speed (17.0 mm/s)
  Call Extruder(1028.16439)
  MoveL 8678 to (468.89, 529.43, 156) mm, rotated rx 180 ry 0 rz 160 deg; joints [10.617, 49.803, 8.243, -145.105, 62.906, 162.377]
  Call Extruder(1031.29610)
  MoveL 8679 to (468.25, 528.74, 156) mm, rotated rx -180 ry 0 rz 160 deg; joints [10.541, 49.689, 8.465, -145.218, 62.971, 162.483]
  Set speed (17.0 mm/s)
  Call Extruder(1034.02772)
  MoveL 8680 to (467.7, 528.12, 156) mm, rotated rx -180 ry 0 rz 160 deg; joints [10.473, 49.592, 8.654, -145.318, 63.026, 162.575]
  Set speed (17.0 mm/s)
  Call Extruder(1036.92977)
  MoveL 8681 to (467.13, 527.45, 156) mm, rotated rx -180 ry 0 rz 160 deg; joints [10.398, 49.49, 8.852, -145.425, 63.083, 162.672]
  Set speed (17.0 mm/s)
  Call Extruder(1039.82899)
  MoveL 8682 to (466.58, 526.77, 156) mm, rotated rx -180 ry 0 rz 160 deg; joints [10.321, 49.39, 9.046, -145.534, 63.137, 162.769]
  Set speed (17.0 mm/s)
  Call Extruder(1042.73178)
  MoveL 8683 to (466.04, 526.09, 156) mm, rotated rx -180 ry 0 rz 160 deg; joints [10.242, 49.292, 9.236, -145.645, 63.19, 162.865]
  Set speed (17.0 mm/s)
  Call Extruder(1045.63567)
  MoveL 8684 to (465.51, 525.38, 156) mm, rotated rx 180 ry 0 rz 160 deg; joints [10.161, 49.196, 9.422, -145.758, 63.241, 162.961]
  Set speed (17.0 mm/s)
  Call Extruder(1048.53876)
  MoveL 8685 to (465, 524.67, 156) mm, rotated rx 180 ry 0 rz 160 deg; joints [10.078, 49.103, 9.603, -145.872, 63.289, 163.057]
  Set speed (17.0 mm/s)
  Call Extruder(1051.41616)
  MoveL 8686 to (464.5, 523.96, 156) mm, rotated rx 180 ry 0 rz 160 deg; joints [9.994, 49.012, 9.78, -145.986, 63.336, 163.151]
  Set speed (17.0 mm/s)
  Call Extruder(1054.53438)
  MoveL 8687 to (463.99, 523.17, 156) mm, rotated rx 180 ry 0 rz 160 deg; joints [9.9, 48.916, 9.965, -146.111, 63.384, 163.252]
  Call Extruder(1060.33728)
  MoveL 8688 to (463.07, 521.68, 156) mm, rotated rx -180 ry 0 rz 160 deg; joints [9.721, 48.745, 10.298, -146.348, 63.466, 163.438]
  Set speed (17.0 mm/s)
  Call Extruder(1063.05579)
  MoveL 8689 to (462.66, 520.97, 156) mm, rotated rx -180 ry 0 rz 160 deg; joints [9.634, 48.668, 10.447, -146.462, 63.502, 163.525]
  Call Extruder(1065.92761)
  MoveL 8690 to (462.25, 520.21, 156) mm, rotated rx 180 ry 0 rz 160 deg; joints [9.54, 48.589, 10.601, -146.582, 63.538, 163.615]
  Set speed (17.0 mm/s)
  Call Extruder(1068.85008)
  MoveL 8691 to (461.84, 519.43, 156) mm, rotated rx -180 ry 0 rz 160 deg; joints [9.444, 48.511, 10.753, -146.706, 63.572, 163.707]
  Set speed (17.0 mm/s)
  Call Extruder(1071.94003)
  MoveL 8692 to (461.42, 518.59, 156) mm, rotated rx -180 ry 0 rz 160 deg; joints [9.34, 48.431, 10.909, -146.838, 63.606, 163.803]
  Set speed (17.0 mm/s)
  Call Extruder(1077.54145)
  MoveL 8693 to (460.72, 517.05, 156) mm, rotated rx 180 ry 0 rz 160 deg; joints [9.146, 48.293, 11.177, -147.081, 63.662, 163.974]
  Set speed (17.0 mm/s)
  Call Extruder(1083.28248)
  MoveL 8694 to (460.06, 515.45, 156) mm, rotated rx 180 ry 0 rz 160 deg; joints [8.942, 48.161, 11.433, -147.333, 63.71, 164.146]
  Set speed (17.0 mm/s)
  Call Extruder(1089.08977)
  MoveL 8695 to (459.46, 513.8, 156) mm, rotated rx -180 ry 0 rz 160 deg; joints [8.729, 48.038, 11.672, -147.592, 63.75, 164.317]
  Set speed (17.0 mm/s)
  Call Extruder(1092.26682)
  MoveL 8696 to (459.17, 512.89, 156) mm, rotated rx -180 ry 0 rz 160 deg; joints [8.61, 47.975, 11.794, -147.735, 63.768, 164.409]
  Set speed (17.0 mm/s)
  Call Extruder(1094.92856)
  MoveL 8697 to (458.93, 512.12, 156) mm, rotated rx -180 ry 0 rz 160 deg; joints [8.51, 47.924, 11.893, -147.856, 63.782, 164.485]
  Set speed (17.0 mm/s)
  Call Extruder(1100.82048)
  MoveL 8698 to (458.46, 510.41, 156) mm, rotated rx 180 ry 0 rz 160 deg; joints [8.284, 47.821, 12.094, -148.124, 63.804, 164.65]
  Set speed (17.0 mm/s)
  Call Extruder(1106.56070)
  MoveL 8699 to (458.08, 508.72, 156) mm, rotated rx -180 ry 0 rz 160 deg; joints [8.059, 47.731, 12.27, -148.388, 63.818, 164.807]
  Set speed (17.0 mm/s)
  Call Extruder(1112.47426)
  MoveL 8700 to (457.75, 506.96, 156) mm, rotated rx 180 ry 0 rz 160 deg; joints [7.823, 47.649, 12.429, -148.662, 63.822, 164.964]
  Set speed (17.0 mm/s)
  Call Extruder(1118.39311)
  MoveL 8701 to (457.49, 505.19, 156) mm, rotated rx -180 ry 0 rz 160 deg; joints [7.583, 47.578, 12.566, -148.937, 63.817, 165.116]
  Set speed (17.0 mm/s)
  Call Extruder(1124.18811)
  MoveL 8702 to (457.32, 503.45, 156) mm, rotated rx -180 ry 0 rz 160 deg; joints [7.345, 47.52, 12.679, -149.207, 63.803, 165.261]
  Set speed (17.0 mm/s)
  Call Extruder(1129.93798)
  MoveL 8703 to (457.21, 501.72, 156) mm, rotated rx -180 ry 0 rz 160 deg; joints [7.106, 47.473, 12.77, -149.476, 63.781, 165.399]
  Set speed (17.0 mm/s)
  Call Extruder(1135.67540)
  MoveL 8704 to (457.18, 499.99, 156) mm, rotated rx -180 ry 0 rz 160 deg; joints [6.867, 47.438, 12.839, -149.743, 63.749, 165.532]
  Set speed (17.0 mm/s)
  Call Extruder(1140.11974)
  MoveL 8705 to (457.2, 498.65, 156) mm, rotated rx 180 ry 0 rz 160 deg; joints [6.68, 47.418, 12.877, -149.949, 63.719, 165.632]
  Set speed (17.0 mm/s)
  Call Extruder(1145.97723)
  MoveL 8706 to (457.29, 496.89, 156) mm, rotated rx 180 ry 0 rz 160 deg; joints [6.433, 47.403, 12.907, -150.22, 63.671, 165.758]
  Set speed (17.0 mm/s)
  Call Extruder(1151.25942)
  MoveL 8707 to (457.44, 495.3, 156) mm, rotated rx 180 ry 0 rz 160 deg; joints [6.21, 47.398, 12.916, -150.462, 63.62, 165.868]
  Call Extruder(1156.60433)
  MoveL 8708 to (457.64, 493.69, 156) mm, rotated rx -180 ry 0 rz 160 deg; joints [5.984, 47.403, 12.906, -150.706, 63.56, 165.974]
  Set speed (17.0 mm/s)
  Call Extruder(1161.79622)
  MoveL 8709 to (457.9, 492.15, 156) mm, rotated rx -180 ry 0 rz 160 deg; joints [5.764, 47.418, 12.878, -150.94, 63.496, 166.073]
  Call Extruder(1166.85446)
  MoveL 8710 to (458.21, 490.65, 156) mm, rotated rx -180 ry 0 rz 160 deg; joints [5.552, 47.44, 12.834, -151.166, 63.426, 166.164]
  Set speed (17.0 mm/s)
  Call Extruder(1172.31703)
  MoveL 8711 to (458.6, 489.05, 156) mm, rotated rx -180 ry 0 rz 160 deg; joints [5.323, 47.475, 12.767, -151.406, 63.343, 166.258]
  Set speed (17.0 mm/s)
  Call Extruder(1177.59326)
  MoveL 8712 to (459.04, 487.52, 156) mm, rotated rx -180 ry 0 rz 160 deg; joints [5.104, 47.517, 12.684, -151.635, 63.256, 166.344]
  Set speed (17.0 mm/s)
  Call Extruder(1182.84251)
  MoveL 8713 to (459.53, 486.01, 156) mm, rotated rx -180 ry 0 rz 160 deg; joints [4.889, 47.569, 12.584, -151.858, 63.162, 166.424]
  Set speed (17.0 mm/s)
  Call Extruder(1187.79425)
  MoveL 8714 to (460.04, 484.61, 156) mm, rotated rx 180 ry 0 rz 160 deg; joints [4.687, 47.626, 12.473, -152.064, 63.067, 166.494]
  Set speed (17.0 mm/s)
  Call Extruder(1193.35176)
  MoveL 8715 to (460.68, 483.05, 156) mm, rotated rx -180 ry 0 rz 160 deg; joints [4.464, 47.7, 12.33, -152.291, 62.954, 166.569]
  Call Extruder(1198.23692)
  MoveL 8716 to (461.28, 481.7, 156) mm, rotated rx -180 ry 0 rz 160 deg; joints [4.271, 47.772, 12.189, -152.486, 62.849, 166.629]
  Set speed (17.0 mm/s)
  Call Extruder(1203.61742)
  MoveL 8717 to (462, 480.25, 156) mm, rotated rx -180 ry 0 rz 160 deg; joints [4.062, 47.861, 12.015, -152.695, 62.726, 166.69]
  Set speed (17.0 mm/s)
  Call Extruder(1208.89816)
  MoveL 8718 to (462.76, 478.85, 156) mm, rotated rx -180 ry 0 rz 160 deg; joints [3.861, 47.958, 11.828, -152.894, 62.599, 166.745]
  Call Extruder(1214.13362)
  MoveL 8719 to (463.57, 477.49, 156) mm, rotated rx -180 ry 0 rz 160 deg; joints [3.666, 48.062, 11.625, -153.085, 62.466, 166.793]
  Call Extruder(1219.11771)
  MoveL 8720 to (464.38, 476.23, 156) mm, rotated rx -180 ry 0 rz 160 deg; joints [3.484, 48.168, 11.418, -153.261, 62.335, 166.834]
  Set speed (17.0 mm/s)
  Call Extruder(1224.57260)
  MoveL 8721 to (465.33, 474.87, 156) mm, rotated rx -180 ry 0 rz 160 deg; joints [3.29, 48.294, 11.174, -153.446, 62.185, 166.873]
  Set speed (17.0 mm/s)
  Call Extruder(1229.89419)
  MoveL 8722 to (466.29, 473.59, 156) mm, rotated rx 180 ry 0 rz 160 deg; joints [3.106, 48.425, 10.919, -153.62, 62.032, 166.906]
  Call Extruder(1234.96531)
  MoveL 8723 to (467.26, 472.4, 156) mm, rotated rx 180 ry 0 rz 160 deg; joints [2.936, 48.558, 10.662, -153.778, 61.882, 166.932]
  Call Extruder(1239.94152)
  MoveL 8724 to (468.25, 471.27, 156) mm, rotated rx 180 ry 0 rz 160 deg; joints [2.774, 48.695, 10.396, -153.927, 61.729, 166.952]
  Call Extruder(1245.33742)
  MoveL 8725 to (469.36, 470.08, 156) mm, rotated rx -180 ry 0 rz 160 deg; joints [2.604, 48.851, 10.092, -154.08, 61.559, 166.967]
  Call Extruder(1250.46621)
  MoveL 8726 to (470.46, 469, 156) mm, rotated rx -180 ry 0 rz 160 deg; joints [2.449, 49.007, 9.789, -154.217, 61.391, 166.977]
  Set speed (17.0 mm/s)
  Call Extruder(1255.83259)
  MoveL 8727 to (471.66, 467.9, 156) mm, rotated rx -180 ry 0 rz 160 deg; joints [2.293, 49.177, 9.458, -154.352, 61.212, 166.98]
  Set speed (17.0 mm/s)
  Call Extruder(1260.98035)
  MoveL 8728 to (472.84, 466.89, 156) mm, rotated rx 180 ry 0 rz 160 deg; joints [2.15, 49.348, 9.127, -154.473, 61.035, 166.978]
  Set speed (17.0 mm/s)
  Call Extruder(1266.33029)
  MoveL 8729 to (474.11, 465.89, 156) mm, rotated rx 180 ry 0 rz 160 deg; joints [2.009, 49.532, 8.77, -154.589, 60.846, 166.969]
  Call Extruder(1271.37317)
  MoveL 8730 to (475.34, 464.99, 156) mm, rotated rx 180 ry 0 rz 160 deg; joints [1.882, 49.712, 8.421, -154.69, 60.665, 166.956]
  Set speed (17.0 mm/s)
  Call Extruder(1276.76787)
  MoveL 8731 to (476.69, 464.08, 156) mm, rotated rx 180 ry 0 rz 160 deg; joints [1.753, 49.911, 8.035, -154.789, 60.466, 166.935]
  Set speed (17.0 mm/s)
  Call Extruder(1281.87547)
  MoveL 8732 to (478, 463.26, 156) mm, rotated rx 180 ry 0 rz 160 deg; joints [1.638, 50.105, 7.658, -154.874, 60.275, 166.909]
  Set speed (17.0 mm/s)
  Call Extruder(1287.17082)
  MoveL 8733 to (479.38, 462.47, 156) mm, rotated rx 180 ry 0 rz 160 deg; joints [1.527, 50.312, 7.256, -154.952, 60.074, 166.876]
  Set speed (17.0 mm/s)
  Call Extruder(1292.46842)
  MoveL 8734 to (480.8, 461.72, 156) mm, rotated rx 180 ry 0 rz 160 deg; joints [1.423, 50.525, 6.843, -155.02, 59.869, 166.837]
  Set speed (17.0 mm/s)
  Call Extruder(1297.50146)
  MoveL 8735 to (482.17, 461.07, 156) mm, rotated rx -180 ry 0 rz 160 deg; joints [1.331, 50.732, 6.442, -155.075, 59.671, 166.794]
  Call Extruder(1302.88807)
  MoveL 8736 to (483.66, 460.42, 156) mm, rotated rx 180 ry 0 rz 160 deg; joints [1.24, 50.959, 6.002, -155.125, 59.457, 166.742]
  Set speed (17.0 mm/s)
  Call Extruder(1308.14099)
  MoveL 8737 to (485.14, 459.84, 156) mm, rotated rx -180 ry 0 rz 160 deg; joints [1.16, 51.185, 5.563, -155.163, 59.246, 166.684]
  Set speed (17.0 mm/s)
  Call Extruder(1313.26503)
  MoveL 8738 to (486.6, 459.33, 156) mm, rotated rx 180 ry 0 rz 160 deg; joints [1.089, 51.41, 5.127, -155.19, 59.038, 166.622]
  Set speed (17.0 mm/s)
  Call Extruder(1318.59077)
  MoveL 8739 to (488.14, 458.85, 156) mm, rotated rx 180 ry 0 rz 160 deg; joints [1.023, 51.648, 4.666, -155.209, 58.82, 166.552]
  Set speed (17.0 mm/s)
  Call Extruder(1323.41724)
  MoveL 8740 to (489.54, 458.48, 156) mm, rotated rx 180 ry 0 rz 160 deg; joints [0.97, 51.867, 4.241, -155.216, 58.621, 166.482]
  Set speed (17.1 mm/s)
  Call Extruder(1328.93066)
  MoveL 8741 to (491.17, 458.1, 156) mm, rotated rx -180 ry 0 rz 160 deg; joints [0.918, 52.122, 3.748, -155.215, 58.392, 166.396]
  Set speed (17.0 mm/s)
  Call Extruder(1333.91783)
  MoveL 8742 to (492.65, 457.81, 156) mm, rotated rx 180 ry 0 rz 160 deg; joints [0.878, 52.355, 3.296, -155.204, 58.185, 166.312]
  Set speed (17.0 mm/s)
  Call Extruder(1339.38589)
  MoveL 8743 to (494.28, 457.56, 156) mm, rotated rx 180 ry 0 rz 160 deg; joints [0.842, 52.614, 2.795, -155.182, 57.956, 166.214]
  Set speed (17.0 mm/s)
  Call Extruder(1344.60489)
  MoveL 8744 to (495.84, 457.38, 156) mm, rotated rx 180 ry 0 rz 160 deg; joints [0.816, 52.863, 2.312, -155.15, 57.738, 166.114]
  Call Extruder(1349.87544)
  MoveL 8745 to (497.43, 457.26, 156) mm, rotated rx -180 ry 0 rz 160 deg; joints [0.797, 53.118, 1.819, -155.108, 57.517, 166.007]
  Set speed (17.0 mm/s)
  Call Extruder(1355.01892)
  MoveL 8746 to (498.98, 457.19, 156) mm, rotated rx -180 ry 0 rz 160 deg; joints [0.786, 53.368, 1.334, -155.058, 57.302, 165.897]
  Call Extruder(1360.26742)
  MoveL 8747 to (500.57, 457.18, 156) mm, rotated rx -180 ry 0 rz 160 deg; joints [0.782, 53.626, 0.836, -154.997, 57.083, 165.778]
  Set speed (17.0 mm/s)
  Call Extruder(1365.23594)
  MoveL 8748 to (502.07, 457.23, 156) mm, rotated rx 180 ry 0 rz 160 deg; joints [0.785, 53.871, 0.362, -154.93, 56.876, 165.661]
  Set speed (17.0 mm/s)
  Call Extruder(1370.71478)
  MoveL 8749 to (503.72, 457.34, 156) mm, rotated rx 180 ry 0 rz 160 deg; joints [0.796, 54.142, -0.163, -154.847, 56.649, 165.525]
  Set speed (17.0 mm/s)
  Call Extruder(1375.91747)
  MoveL 8750 to (505.28, 457.51, 156) mm, rotated rx -180 ry 0 rz 160 deg; joints [0.814, 54.4, -0.663, -154.758, 56.435, 165.39]
  Call Extruder(1380.89536)
  MoveL 8751 to (506.77, 457.72, 156) mm, rotated rx -180 ry 0 rz 160 deg; joints [0.838, 54.648, -1.141, -154.664, 56.232, 165.256]
  Set speed (17.0 mm/s)
  Call Extruder(1386.27355)
  MoveL 8752 to (508.37, 458, 156) mm, rotated rx 180 ry 0 rz 160 deg; joints [0.871, 54.916, -1.659, -154.554, 56.015, 165.106]
  Call Extruder(1391.56901)
  MoveL 8753 to (509.93, 458.35, 156) mm, rotated rx 180 ry 0 rz 160 deg; joints [0.911, 55.179, -2.168, -154.436, 55.803, 164.952]
  Set speed (17.0 mm/s)
  Call Extruder(1397.13839)
  MoveL 8754 to (511.56, 458.76, 156) mm, rotated rx -180 ry 0 rz 160 deg; joints [0.96, 55.456, -2.702, -154.303, 55.584, 164.785]
  Set speed (17.0 mm/s)
  Call Extruder(1400.35100)
  MoveL 8755 to (512.49, 459.05, 156) mm, rotated rx 180 ry 0 rz 160 deg; joints [0.993, 55.614, -3.009, -154.22, 55.459, 164.685]
  Set speed (17.0 mm/s)
  Call Extruder(1401.31897)
  MoveL 8756 to (512.77, 459.12, 156) mm, rotated rx -180 ry 0 rz 160 deg; joints [1.002, 55.663, -3.102, -154.196, 55.421, 164.655]
  Set speed (17.0 mm/s)
  Call Extruder(1407.29412)
  MoveL 8757 to (514.48, 459.7, 156) mm, rotated rx 180 ry 0 rz 160 deg; joints [1.069, 55.957, -3.67, -154.034, 55.192, 164.465]
  Set speed (17.0 mm/s)
  Call Extruder(1412.18085)
  MoveL 8758 to (515.86, 460.22, 156) mm, rotated rx -180 ry 0 rz 160 deg; joints [1.131, 56.196, -4.132, -153.894, 55.009, 164.304]
  Call Extruder(1417.70236)
  MoveL 8759 to (517.39, 460.87, 156) mm, rotated rx 180 ry 0 rz 160 deg; joints [1.206, 56.464, -4.65, -153.727, 54.805, 164.118]
  Set speed (17.0 mm/s)
  Call Extruder(1422.93408)
  MoveL 8760 to (518.83, 461.54, 156) mm, rotated rx -180 ry 0 rz 160 deg; joints [1.285, 56.716, -5.137, -153.561, 54.617, 163.938]
  Set speed (17.0 mm/s)
  Call Extruder(1427.89124)
  MoveL 8761 to (520.16, 462.22, 156) mm, rotated rx 180 ry 0 rz 160 deg; joints [1.364, 56.952, -5.593, -153.398, 54.442, 163.763]
  Set speed (17.0 mm/s)
  Call Extruder(1433.36370)
  MoveL 8762 to (521.6, 463.03, 156) mm, rotated rx 180 ry 0 rz 160 deg; joints [1.458, 57.21, -6.09, -153.21, 54.254, 163.565]
  Set speed (17.0 mm/s)
  Call Extruder(1438.54685)
  MoveL 8763 to (522.94, 463.84, 156) mm, rotated rx -180 ry 0 rz 160 deg; joints [1.552, 57.451, -6.555, -153.025, 54.081, 163.375]
  Set speed (17.0 mm/s)
  Call Extruder(1443.69818)
  MoveL 8764 to (524.24, 464.7, 156) mm, rotated rx -180 ry 0 rz 160 deg; joints [1.652, 57.687, -7.01, -152.835, 53.915, 163.183]
  Set speed (17.0 mm/s)
  Call Extruder(1448.82815)
  MoveL 8765 to (525.5, 465.6, 156) mm, rotated rx 180 ry 0 rz 160 deg; joints [1.756, 57.917, -7.456, -152.64, 53.754, 162.988]
  Set speed (17.0 mm/s)
  Call Extruder(1454.25162)
  MoveL 8766 to (526.79, 466.6, 156) mm, rotated rx -180 ry 0 rz 160 deg; joints [1.871, 58.157, -7.918, -152.427, 53.591, 162.78]
  Set speed (17.0 mm/s)
  Call Extruder(1459.51135)
  MoveL 8767 to (528.01, 467.61, 156) mm, rotated rx 180 ry 0 rz 160 deg; joints [1.988, 58.385, -8.357, -152.215, 53.438, 162.575]
  Set speed (17.0 mm/s)
  Call Extruder(1464.66944)
  MoveL 8768 to (529.18, 468.65, 156) mm, rotated rx -180 ry 0 rz 160 deg; joints [2.108, 58.603, -8.779, -152.003, 53.295, 162.372]
  Set speed (17.0 mm/s)
  Call Extruder(1469.87147)
  MoveL 8769 to (530.3, 469.75, 156) mm, rotated rx 180 ry 0 rz 160 deg; joints [2.233, 58.818, -9.193, -151.784, 53.157, 162.165]
  Set speed (17.0 mm/s)
  Call Extruder(1472.55359)
  MoveL 8770 to (530.87, 470.32, 156) mm, rotated rx -180 ry 0 rz 160 deg; joints [2.3, 58.927, -9.402, -151.669, 53.089, 162.058]
  Call Extruder(1475.44297)
  MoveL 8771 to (531.47, 470.96, 156) mm, rotated rx 180 ry 0 rz 160 deg; joints [2.372, 59.042, -9.624, -151.544, 53.018, 161.943]
  Set speed (17.0 mm/s)
  Call Extruder(1478.35163)
  MoveL 8772 to (532.06, 471.61, 156) mm, rotated rx 180 ry 0 rz 160 deg; joints [2.447, 59.156, -9.844, -151.417, 52.948, 161.826]
  Set speed (17.0 mm/s)
  Call Extruder(1481.18908)
  MoveL 8773 to (532.62, 472.26, 156) mm, rotated rx -180 ry 0 rz 160 deg; joints [2.521, 59.266, -10.056, -151.293, 52.881, 161.712]
  Set speed (17.1 mm/s)
  Call Extruder(1484.14542)
  MoveL 8774 to (533.19, 472.94, 156) mm, rotated rx -180 ry 0 rz 160 deg; joints [2.599, 59.378, -10.272, -151.161, 52.815, 161.593]
  Set speed (17.0 mm/s)
  Call Extruder(1487.08474)
  MoveL 8775 to (533.75, 473.64, 156) mm, rotated rx 180 ry 0 rz 160 deg; joints [2.678, 59.488, -10.483, -151.03, 52.751, 161.474]
  Set speed (17.0 mm/s)
  Call Extruder(1489.98409)
  MoveL 8776 to (534.28, 474.33, 156) mm, rotated rx -180 ry 0 rz 160 deg; joints [2.757, 59.593, -10.687, -150.899, 52.691, 161.357]
  Set speed (17.0 mm/s)
  Call Extruder(1493.06290)
  MoveL 8777 to (534.82, 475.08, 156) mm, rotated rx 180 ry 0 rz 160 deg; joints [2.843, 59.703, -10.898, -150.759, 52.629, 161.233]
  Call Extruder(1495.72366)
  MoveL 8778 to (535.29, 475.74, 156) mm, rotated rx 180 ry 0 rz 160 deg; joints [2.918, 59.797, -11.078, -150.638, 52.578, 161.125]
  Set speed (17.0 mm/s)
  Call Extruder(1498.61513)
  MoveL 8779 to (535.77, 476.46, 156) mm, rotated rx 180 ry 0 rz 160 deg; joints [3, 59.896, -11.269, -150.505, 52.525, 161.009]
  Call Extruder(1501.75486)
  MoveL 8780 to (536.29, 477.26, 156) mm, rotated rx 180 ry 0 rz 160 deg; joints [3.091, 60.001, -11.472, -150.36, 52.469, 160.882]
  Set speed (17.0 mm/s)
  Call Extruder(1504.53454)
  MoveL 8781 to (536.73, 477.98, 156) mm, rotated rx -180 ry 0 rz 160 deg; joints [3.172, 60.091, -11.646, -150.231, 52.423, 160.771]
  Call Extruder(1507.52338)
  MoveL 8782 to (537.18, 478.76, 156) mm, rotated rx -180 ry 0 rz 160 deg; joints [3.26, 60.187, -11.83, -150.092, 52.376, 160.651]
  Set speed (17.0 mm/s)
  Call Extruder(1512.12138)
  MoveL 8783 to (537.85, 479.97, 156) mm, rotated rx -180 ry 0 rz 160 deg; joints [3.398, 60.328, -12.103, -149.878, 52.308, 160.468]
  Set speed (17.0 mm/s)
  Call Extruder(1515.42960)
  MoveL 8784 to (538.31, 480.86, 156) mm, rotated rx 180 ry 0 rz 160 deg; joints [3.499, 60.426, -12.291, -149.722, 52.264, 160.337]
  Set speed (17.1 mm/s)
  Call Extruder(1519.02515)
  MoveL 8785 to (538.78, 481.84, 156) mm, rotated rx 180 ry 0 rz 160 deg; joints [3.61, 60.528, -12.487, -149.553, 52.22, 160.196]
  Set speed (17.0 mm/s)
  Call Extruder(1522.05911)
  MoveL 8786 to (539.16, 482.67, 156) mm, rotated rx 180 ry 0 rz 160 deg; joints [3.705, 60.611, -12.648, -149.41, 52.186, 160.077]
  Set speed (17.0 mm/s)
  Call Extruder(1527.65468)
  MoveL 8787 to (539.81, 484.23, 156) mm, rotated rx 180 ry 0 rz 160 deg; joints [3.882, 60.757, -12.928, -149.146, 52.13, 159.861]
  Call Extruder(1533.44983)
  MoveL 8788 to (540.42, 485.87, 156) mm, rotated rx -180 ry 0 rz 160 deg; joints [4.068, 60.898, -13.199, -148.873, 52.083, 159.64]
  Call Extruder(1539.26458)
  MoveL 8789 to (540.97, 487.54, 156) mm, rotated rx -180 ry 0 rz 160 deg; joints [4.257, 61.028, -13.449, -148.599, 52.047, 159.423]
  Set speed (17.0 mm/s)
  Call Extruder(1542.36895)
  MoveL 8790 to (541.23, 488.44, 156) mm, rotated rx -180 ry 0 rz 160 deg; joints [4.36, 61.091, -13.572, -148.453, 52.033, 159.309]
  Set speed (17.0 mm/s)
  Call Extruder(1545.27153)
  MoveL 8791 to (541.46, 489.28, 156) mm, rotated rx -180 ry 0 rz 160 deg; joints [4.456, 61.149, -13.683, -148.318, 52.021, 159.203]
  Set speed (17.0 mm/s)
  Call Extruder(1550.84410)
  MoveL 8792 to (541.85, 490.92, 156) mm, rotated rx 180 ry 0 rz 160 deg; joints [4.642, 61.251, -13.878, -148.058, 52.008, 159.005]
  Call Extruder(1556.73333)
  MoveL 8793 to (542.19, 492.67, 156) mm, rotated rx -180 ry 0 rz 160 deg; joints [4.841, 61.346, -14.062, -147.786, 52.005, 158.8]
  Set speed (17.0 mm/s)
  Call Extruder(1562.78096)
  MoveL 8794 to (542.46, 494.47, 156) mm, rotated rx 180 ry 0 rz 160 deg; joints [5.047, 61.431, -14.225, -147.51, 52.013, 158.597]
  Set speed (17.0 mm/s)
  Call Extruder(1568.53077)
  MoveL 8795 to (542.65, 496.2, 156) mm, rotated rx 180 ry 0 rz 160 deg; joints [5.244, 61.499, -14.356, -147.25, 52.033, 158.411]
  Call Extruder(0.00000)
  Set speed (17.0 mm/s)
  Call Extruder(5.60818)
  MoveL 8796 to (542.77, 497.89, 156) mm, rotated rx 180 ry 0 rz 160 deg; joints [5.438, 61.553, -14.46, -147.001, 52.062, 158.236]
  Set speed (17.0 mm/s)
  Call Extruder(11.39765)
  MoveL 8797 to (542.82, 499.63, 156) mm, rotated rx 180 ry 0 rz 160 deg; joints [5.639, 61.596, -14.543, -146.747, 52.104, 158.063]
  Set speed (17.0 mm/s)
  Call Extruder(17.42254)
  MoveL 8798 to (542.8, 501.45, 156) mm, rotated rx 180 ry 0 rz 160 deg; joints [5.849, 61.628, -14.604, -146.488, 52.158, 157.891]
  Set speed (17.0 mm/s)
  Call Extruder(23.19352)
  MoveL 8799 to (542.7, 503.19, 156) mm, rotated rx 180 ry 0 rz 160 deg; joints [6.051, 61.645, -14.637, -146.245, 52.221, 157.735]
  Call Extruder(29.03672)
  MoveL 8800 to (542.53, 504.95, 156) mm, rotated rx 180 ry 0 rz 160 deg; joints [6.255, 61.649, -14.644, -146.004, 52.296, 157.586]
  Call Extruder(34.70192)
  MoveL 8801 to (542.3, 506.65, 156) mm, rotated rx 180 ry 0 rz 160 deg; joints [6.453, 61.641, -14.629, -145.776, 52.378, 157.45]
  Set speed (17.0 mm/s)
  Call Extruder(40.39142)
  MoveL 8802 to (542, 508.34, 156) mm, rotated rx 180 ry 0 rz 160 deg; joints [6.652, 61.62, -14.589, -145.553, 52.47, 157.323]
  Set speed (17.0 mm/s)
  Call Extruder(46.37908)
  MoveL 8803 to (541.61, 510.1, 156) mm, rotated rx -180 ry 0 rz 160 deg; joints [6.86, 61.584, -14.52, -145.325, 52.577, 157.199]
  Set speed (17.0 mm/s)
  Call Extruder(52.01574)
  MoveL 8804 to (541.18, 511.75, 156) mm, rotated rx 180 ry 0 rz 160 deg; joints [7.056, 61.539, -14.432, -145.117, 52.688, 157.092]
  Set speed (17.0 mm/s)
  Call Extruder(57.93874)
  MoveL 8805 to (540.65, 513.46, 156) mm, rotated rx -180 ry 0 rz 160 deg; joints [7.26, 61.477, -14.314, -144.906, 52.814, 156.989]
  Set speed (17.0 mm/s)
  Call Extruder(63.53240)
  MoveL 8806 to (540.09, 515.05, 156) mm, rotated rx 180 ry 0 rz 160 deg; joints [7.452, 61.407, -14.179, -144.713, 52.942, 156.903]
  Set speed (17.0 mm/s)
  Call Extruder(66.64735)
  MoveL 8807 to (539.75, 515.93, 156) mm, rotated rx 180 ry 0 rz 160 deg; joints [7.558, 61.363, -14.094, -144.609, 53.017, 156.859]
  Set speed (17.0 mm/s)
  Call Extruder(69.54196)
  MoveL 8808 to (539.42, 516.74, 156) mm, rotated rx -180 ry 0 rz 160 deg; joints [7.656, 61.32, -14.011, -144.513, 53.089, 156.82]
  Set speed (17.0 mm/s)
  Call Extruder(75.11365)
  MoveL 8809 to (538.73, 518.27, 156) mm, rotated rx 180 ry 0 rz 160 deg; joints [7.844, 61.226, -13.832, -144.335, 53.233, 156.754]
  Set speed (17.0 mm/s)
  Call Extruder(78.13436)
  MoveL 8810 to (538.33, 519.09, 156) mm, rotated rx -180 ry 0 rz 160 deg; joints [7.944, 61.171, -13.724, -144.242, 53.314, 156.722]
  Set speed (17.0 mm/s)
  Call Extruder(81.11297)
  MoveL 8811 to (537.92, 519.89, 156) mm, rotated rx 180 ry 0 rz 160 deg; joints [8.043, 61.113, -13.614, -144.152, 53.396, 156.693]
  Set speed (17.0 mm/s)
  Call Extruder(83.83104)
  MoveL 8812 to (537.53, 520.62, 156) mm, rotated rx 180 ry 0 rz 160 deg; joints [8.133, 61.058, -13.507, -144.071, 53.473, 156.669]
  Set speed (17.0 mm/s)
  Call Extruder(86.90380)
  MoveL 8813 to (537.08, 521.42, 156) mm, rotated rx -180 ry 0 rz 160 deg; joints [8.234, 60.992, -13.381, -143.983, 53.563, 156.645]
  Set speed (17.0 mm/s)
  Call Extruder(89.62448)
  MoveL 8814 to (536.66, 522.13, 156) mm, rotated rx 180 ry 0 rz 160 deg; joints [8.323, 60.932, -13.265, -143.906, 53.643, 156.626]
  Set speed (17.0 mm/s)
  Call Extruder(92.59364)
  MoveL 8815 to (536.19, 522.89, 156) mm, rotated rx 180 ry 0 rz 160 deg; joints [8.419, 60.863, -13.131, -143.824, 53.733, 156.608]
  Set speed (17.0 mm/s)
  Call Extruder(95.46893)
  MoveL 8816 to (535.72, 523.62, 156) mm, rotated rx 180 ry 0 rz 160 deg; joints [8.511, 60.793, -12.996, -143.747, 53.822, 156.594]
  Set speed (17.0 mm/s)
  Call Extruder(98.38963)
  MoveL 8817 to (535.23, 524.35, 156) mm, rotated rx -180 ry 0 rz 160 deg; joints [8.604, 60.719, -12.855, -143.671, 53.913, 156.581]
  Set speed (17.0 mm/s)
  Call Extruder(101.21982)
  MoveL 8818 to (534.73, 525.05, 156) mm, rotated rx 180 ry 0 rz 160 deg; joints [8.693, 60.645, -12.712, -143.599, 54.004, 156.572]
  Call Extruder(104.34834)
  MoveL 8819 to (534.17, 525.81, 156) mm, rotated rx -180 ry 0 rz 160 deg; joints [8.791, 60.56, -12.549, -143.522, 54.106, 156.564]
  Set speed (17.0 mm/s)
  Call Extruder(107.23186)
  MoveL 8820 to (533.64, 526.5, 156) mm, rotated rx 180 ry 0 rz 160 deg; joints [8.881, 60.479, -12.393, -143.453, 54.202, 156.56]
  Set speed (17.0 mm/s)
  Call Extruder(110.00373)
  MoveL 8821 to (533.12, 527.15, 156) mm, rotated rx 180 ry 0 rz 160 deg; joints [8.966, 60.4, -12.24, -143.388, 54.295, 156.558]
  Set speed (17.0 mm/s)
  Call Extruder(113.99072)
  MoveL 8822 to (532.34, 528.07, 156) mm, rotated rx 180 ry 0 rz 160 deg; joints [9.087, 60.281, -12.01, -143.299, 54.432, 156.559]
  Set speed (17.0 mm/s)
  Call Extruder(118.72158)
  MoveL 8823 to (531.38, 529.13, 156) mm, rotated rx 180 ry 0 rz 160 deg; joints [9.228, 60.133, -11.725, -143.198, 54.597, 156.568]
  Set speed (17.0 mm/s)
  Call Extruder(121.54646)
  MoveL 8824 to (530.8, 529.75, 156) mm, rotated rx -180 ry 0 rz 160 deg; joints [9.311, 60.041, -11.55, -143.141, 54.698, 156.576]
  Call Extruder(124.44993)
  MoveL 8825 to (530.18, 530.38, 156) mm, rotated rx 180 ry 0 rz 160 deg; joints [9.395, 59.946, -11.365, -143.084, 54.803, 156.586]
  Call Extruder(127.38877)
  MoveL 8826 to (529.55, 531, 156) mm, rotated rx 180 ry 0 rz 160 deg; joints [9.48, 59.846, -11.173, -143.028, 54.91, 156.6]
  Set speed (17.0 mm/s)
  Call Extruder(130.30614)
  MoveL 8827 to (528.9, 531.6, 156) mm, rotated rx -180 ry 0 rz 160 deg; joints [9.562, 59.745, -10.978, -142.975, 55.018, 156.615]
  Set speed (17.1 mm/s)
  Call Extruder(134.49846)
  MoveL 8828 to (527.96, 532.44, 156) mm, rotated rx 180 ry 0 rz 160 deg; joints [9.679, 59.596, -10.691, -142.902, 55.174, 156.642]
  Set speed (17.1 mm/s)
  Call Extruder(139.02047)
  MoveL 8829 to (526.91, 533.31, 156) mm, rotated rx -180 ry 0 rz 160 deg; joints [9.802, 59.429, -10.37, -142.83, 55.346, 156.677]
  Set speed (17.0 mm/s)
  Call Extruder(141.81873)
  MoveL 8830 to (526.25, 533.84, 156) mm, rotated rx -180 ry 0 rz 160 deg; joints [9.877, 59.324, -10.168, -142.787, 55.453, 156.701]
  Call Extruder(144.77158)
  MoveL 8831 to (525.53, 534.38, 156) mm, rotated rx -180 ry 0 rz 160 deg; joints [9.955, 59.211, -9.95, -142.744, 55.567, 156.729]
  Call Extruder(147.70748)
  MoveL 8832 to (524.82, 534.9, 156) mm, rotated rx -180 ry 0 rz 160 deg; joints [10.03, 59.097, -9.73, -142.703, 55.682, 156.759]
  Set speed (17.0 mm/s)
  Call Extruder(150.58623)
  MoveL 8833 to (524.1, 535.39, 156) mm, rotated rx 180 ry 0 rz 160 deg; joints [10.103, 58.983, -9.51, -142.666, 55.795, 156.791]
  Set speed (17.0 mm/s)
  Call Extruder(153.45948)
  MoveL 8834 to (523.38, 535.88, 156) mm, rotated rx 180 ry 0 rz 160 deg; joints [10.175, 58.867, -9.287, -142.63, 55.908, 156.825]
  Set speed (17.0 mm/s)
  Call Extruder(155.70658)
  MoveL 8835 to (522.81, 536.24, 156) mm, rotated rx -180 ry 0 rz 160 deg; joints [10.23, 58.775, -9.11, -142.604, 55.997, 156.853]
  Set speed (17.0 mm/s)
  Call Extruder(160.16908)
  MoveL 8836 to (521.66, 536.94, 156) mm, rotated rx -180 ry 0 rz 160 deg; joints [10.337, 58.591, -8.754, -142.555, 56.175, 156.913]
  Set speed (17.0 mm/s)
  Call Extruder(164.98965)
  MoveL 8837 to (520.39, 537.66, 156) mm, rotated rx 180 ry 0 rz 160 deg; joints [10.449, 58.386, -8.36, -142.509, 56.37, 156.983]
  Set speed (17.0 mm/s)
  Call Extruder(167.95349)
  MoveL 8838 to (519.6, 538.07, 156) mm, rotated rx -180 ry 0 rz 160 deg; joints [10.515, 58.258, -8.113, -142.484, 56.49, 157.029]
  Set speed (17.0 mm/s)
  Call Extruder(171.10535)
  MoveL 8839 to (518.75, 538.5, 156) mm, rotated rx 180 ry 0 rz 160 deg; joints [10.585, 58.121, -7.849, -142.458, 56.618, 157.08]
  Set speed (17.0 mm/s)
  Call Extruder(174.03331)
  MoveL 8840 to (517.95, 538.88, 156) mm, rotated rx 180 ry 0 rz 160 deg; joints [10.647, 57.992, -7.599, -142.438, 56.737, 157.129]
  Set speed (17.0 mm/s)
  Call Extruder(179.80775)
  MoveL 8841 to (516.35, 539.58, 156) mm, rotated rx 180 ry 0 rz 160 deg; joints [10.766, 57.733, -7.1, -142.403, 56.974, 157.233]
  Set speed (17.0 mm/s)
  Call Extruder(185.61201)
  MoveL 8842 to (514.72, 540.21, 156) mm, rotated rx 180 ry 0 rz 160 deg; joints [10.878, 57.468, -6.589, -142.376, 57.212, 157.345]
  Set speed (17.0 mm/s)
  Call Extruder(188.00076)
  MoveL 8843 to (514.04, 540.45, 156) mm, rotated rx -180 ry 0 rz 160 deg; joints [10.923, 57.358, -6.376, -142.368, 57.311, 157.393]
  Set speed (17.0 mm/s)
  Call Extruder(191.43004)
  MoveL 8844 to (513.06, 540.78, 156) mm, rotated rx 180 ry 0 rz 160 deg; joints [10.985, 57.199, -6.069, -142.358, 57.452, 157.464]
  Set speed (17.0 mm/s)
  Call Extruder(196.59223)
  MoveL 8845 to (511.57, 541.24, 156) mm, rotated rx -180 ry 0 rz 160 deg; joints [11.073, 56.956, -5.6, -142.348, 57.665, 157.575]
  Set speed (17.0 mm/s)
  Call Extruder(203.02677)
  MoveL 8846 to (509.69, 541.71, 156) mm, rotated rx 180 ry 0 rz 160 deg; joints [11.175, 56.648, -5.006, -142.347, 57.93, 157.723]
  Call Extruder(208.68742)
  MoveL 8847 to (508.01, 542.07, 156) mm, rotated rx -180 ry 0 rz 160 deg; joints [11.257, 56.375, -4.479, -142.354, 58.162, 157.858]
  Call Extruder(214.56399)
  MoveL 8848 to (506.27, 542.36, 156) mm, rotated rx 180 ry 0 rz 160 deg; joints [11.335, 56.089, -3.926, -142.37, 58.403, 158.005]
  Set speed (17.0 mm/s)
  Call Extruder(220.50240)
  MoveL 8849 to (504.49, 542.59, 156) mm, rotated rx 180 ry 0 rz 160 deg; joints [11.406, 55.797, -3.363, -142.395, 58.644, 158.159]
  Call Extruder(226.27274)
  MoveL 8850 to (502.75, 542.73, 156) mm, rotated rx 180 ry 0 rz 160 deg; joints [11.466, 55.512, -2.812, -142.427, 58.877, 158.315]
  Set speed (17.0 mm/s)
  Call Extruder(231.95962)
  MoveL 8851 to (501.04, 542.81, 156) mm, rotated rx 180 ry 0 rz 160 deg; joints [11.518, 55.23, -2.267, -142.467, 59.105, 158.473]
  Call Extruder(237.58434)
  MoveL 8852 to (499.34, 542.82, 156) mm, rotated rx 180 ry 0 rz 160 deg; joints [11.562, 54.951, -1.727, -142.515, 59.328, 158.634]
  Set speed (10.0 mm/s)
  MoveL 8853 to (499.34, 542.82, 160) mm, rotated rx -180 ry 0 rz 160 deg; joints [11.562, 54.387, -1.605, -142.354, 58.977, 158.32]
  Set speed (120.0 mm/s)
  MoveL 8854 to (499.36, 541.49, 160) mm, rotated rx -180 ry 0 rz 160 deg; joints [11.398, 54.346, -1.526, -142.546, 58.947, 158.438]
  Set speed (17.1 mm/s)
  Call Extruder(243.32683)
  MoveL 8855 to (497.62, 541.42, 160) mm, rotated rx -180 ry 0 rz 160 deg; joints [11.433, 54.057, -0.971, -142.604, 59.171, 158.607]
  Set speed (17.1 mm/s)
  Call Extruder(248.95165)
  MoveL 8856 to (495.92, 541.29, 160) mm, rotated rx 180 ry 0 rz 160 deg; joints [11.459, 53.775, -0.428, -142.67, 59.388, 158.776]
  Call Extruder(254.47345)
  MoveL 8857 to (494.25, 541.09, 160) mm, rotated rx 180 ry 0 rz 160 deg; joints [11.477, 53.498, 0.104, -142.742, 59.597, 158.946]
  Set speed (17.1 mm/s)
  Call Extruder(260.03663)
  MoveL 8858 to (492.59, 540.82, 160) mm, rotated rx -180 ry 0 rz 160 deg; joints [11.485, 53.219, 0.638, -142.824, 59.804, 159.121]
  Set speed (17.1 mm/s)
  Call Extruder(265.77018)
  MoveL 8859 to (490.88, 540.48, 160) mm, rotated rx -180 ry 0 rz 160 deg; joints [11.485, 52.934, 1.187, -142.916, 60.014, 159.305]
  Set speed (17.1 mm/s)
  Call Extruder(271.33254)
  MoveL 8860 to (489.25, 540.07, 160) mm, rotated rx 180 ry 0 rz 160 deg; joints [11.476, 52.659, 1.715, -143.013, 60.213, 159.485]
  Set speed (17.1 mm/s)
  Call Extruder(276.77801)
  MoveL 8861 to (487.66, 539.61, 160) mm, rotated rx -180 ry 0 rz 160 deg; joints [11.459, 52.393, 2.227, -143.116, 60.403, 159.665]
  Set speed (17.1 mm/s)
  Call Extruder(282.38698)
  MoveL 8862 to (486.05, 539.08, 160) mm, rotated rx 180 ry 0 rz 160 deg; joints [11.432, 52.12, 2.751, -143.23, 60.595, 159.852]
  Set speed (17.1 mm/s)
  Call Extruder(288.29855)
  MoveL 8863 to (484.37, 538.44, 160) mm, rotated rx 180 ry 0 rz 160 deg; joints [11.394, 51.837, 3.295, -143.358, 60.792, 160.051]
  Set speed (17.1 mm/s)
  Call Extruder(293.71240)
  MoveL 8864 to (482.86, 537.79, 160) mm, rotated rx 180 ry 0 rz 160 deg; joints [11.35, 51.581, 3.788, -143.484, 60.966, 160.235]
  Set speed (17.1 mm/s)
  Call Extruder(296.64945)
  MoveL 8865 to (482.06, 537.41, 160) mm, rotated rx -180 ry 0 rz 160 deg; joints [11.323, 51.444, 4.052, -143.555, 61.059, 160.336]
  Set speed (17.1 mm/s)
  Call Extruder(300.45269)
  MoveL 8866 to (481.02, 536.9, 160) mm, rotated rx 180 ry 0 rz 160 deg; joints [11.284, 51.267, 4.391, -143.65, 61.177, 160.466]
  Set speed (17.1 mm/s)
  Call Extruder(305.09040)
  MoveL 8867 to (479.78, 536.23, 160) mm, rotated rx 180 ry 0 rz 160 deg; joints [11.23, 51.055, 4.798, -143.772, 61.317, 160.626]
  Set speed (17.1 mm/s)
  Call Extruder(307.54933)
  MoveL 8868 to (479.14, 535.87, 160) mm, rotated rx -180 ry 0 rz 160 deg; joints [11.199, 50.944, 5.012, -143.838, 61.389, 160.711]
  Set speed (17.1 mm/s)
  Call Extruder(310.82129)
  MoveL 8869 to (478.28, 535.35, 160) mm, rotated rx 180 ry 0 rz 160 deg; joints [11.155, 50.798, 5.294, -143.929, 61.484, 160.825]
  Set speed (17.1 mm/s)
  Call Extruder(313.22507)
  MoveL 8870 to (477.67, 534.97, 160) mm, rotated rx 180 ry 0 rz 160 deg; joints [11.12, 50.691, 5.499, -143.998, 61.552, 160.908]
  Set speed (17.1 mm/s)
  Call Extruder(316.25949)
  MoveL 8871 to (476.9, 534.46, 160) mm, rotated rx 180 ry 0 rz 160 deg; joints [11.075, 50.558, 5.755, -144.086, 61.637, 161.013]
  Set speed (17.1 mm/s)
  Call Extruder(318.86657)
  MoveL 8872 to (476.24, 534.02, 160) mm, rotated rx 180 ry 0 rz 160 deg; joints [11.034, 50.445, 5.972, -144.163, 61.708, 161.104]
  Call Extruder(324.46845)
  MoveL 8873 to (474.87, 533.02, 160) mm, rotated rx 180 ry 0 rz 160 deg; joints [10.938, 50.207, 6.431, -144.335, 61.856, 161.299]
  Call Extruder(327.26255)
  MoveL 8874 to (474.2, 532.5, 160) mm, rotated rx 180 ry 0 rz 160 deg; joints [10.887, 50.09, 6.656, -144.423, 61.928, 161.396]
  Set speed (17.1 mm/s)
  Call Extruder(330.03730)
  MoveL 8875 to (473.55, 531.97, 160) mm, rotated rx -180 ry 0 rz 160 deg; joints [10.835, 49.975, 6.876, -144.512, 61.997, 161.492]
  Set speed (17.1 mm/s)
  Call Extruder(333.73521)
  MoveL 8876 to (472.69, 531.24, 160) mm, rotated rx -180 ry 0 rz 160 deg; joints [10.761, 49.825, 7.165, -144.634, 62.087, 161.62]
  Set speed (17.1 mm/s)
  Call Extruder(338.40415)
  MoveL 8877 to (471.64, 530.29, 160) mm, rotated rx -180 ry 0 rz 160 deg; joints [10.662, 49.64, 7.521, -144.792, 62.195, 161.781]
  Set speed (17.1 mm/s)
  Call Extruder(340.73208)
  MoveL 8878 to (471.13, 529.8, 160) mm, rotated rx 180 ry 0 rz 160 deg; joints [10.611, 49.55, 7.696, -144.873, 62.248, 161.862]
  Set speed (17.1 mm/s)
  Call Extruder(343.97718)
  MoveL 8879 to (470.43, 529.11, 160) mm, rotated rx -180 ry 0 rz 160 deg; joints [10.537, 49.425, 7.934, -144.987, 62.319, 161.973]
  Set speed (17.1 mm/s)
  Call Extruder(346.84068)
  MoveL 8880 to (469.83, 528.48, 160) mm, rotated rx 180 ry 0 rz 160 deg; joints [10.469, 49.318, 8.141, -145.09, 62.379, 162.071]
  Set speed (17.1 mm/s)
  Call Extruder(349.63513)
  MoveL 8881 to (469.25, 527.86, 160) mm, rotated rx 180 ry 0 rz 160 deg; joints [10.4, 49.214, 8.34, -145.192, 62.437, 162.167]
  Set speed (17.1 mm/s)
  Call Extruder(352.64373)
  MoveL 8882 to (468.65, 527.18, 160) mm, rotated rx -180 ry 0 rz 160 deg; joints [10.324, 49.105, 8.55, -145.303, 62.496, 162.269]
  Set speed (17.1 mm/s)
  Call Extruder(355.51236)
  MoveL 8883 to (468.09, 526.52, 160) mm, rotated rx 180 ry 0 rz 160 deg; joints [10.25, 49.003, 8.747, -145.411, 62.551, 162.367]
  Set speed (17.1 mm/s)
  Call Extruder(358.02409)
  MoveL 8884 to (467.6, 525.92, 160) mm, rotated rx 180 ry 0 rz 160 deg; joints [10.183, 48.916, 8.915, -145.507, 62.598, 162.452]
  Call Extruder(360.83185)
  MoveL 8885 to (467.08, 525.25, 160) mm, rotated rx 180 ry 0 rz 160 deg; joints [10.106, 48.82, 9.099, -145.616, 62.648, 162.546]
  Set speed (17.1 mm/s)
  Call Extruder(363.95609)
  MoveL 8886 to (466.51, 524.5, 160) mm, rotated rx -180 ry 0 rz 160 deg; joints [10.018, 48.716, 9.3, -145.738, 62.701, 162.65]
  Set speed (17.1 mm/s)
  Call Extruder(366.32575)
  MoveL 8887 to (466.09, 523.91, 160) mm, rotated rx -180 ry 0 rz 160 deg; joints [9.95, 48.639, 9.449, -145.832, 62.74, 162.729]
  Call Extruder(371.96119)
  MoveL 8888 to (465.13, 522.49, 160) mm, rotated rx 180 ry 0 rz 160 deg; joints [9.782, 48.461, 9.791, -146.059, 62.826, 162.915]
  Set speed (17.1 mm/s)
  Call Extruder(374.82121)
  MoveL 8889 to (464.67, 521.76, 160) mm, rotated rx -180 ry 0 rz 160 deg; joints [9.694, 48.374, 9.958, -146.177, 62.867, 163.009]
  Set speed (17.1 mm/s)
  Call Extruder(377.62906)
  MoveL 8890 to (464.23, 521.03, 160) mm, rotated rx -180 ry 0 rz 160 deg; joints [9.606, 48.291, 10.118, -146.294, 62.906, 163.1]
  Call Extruder(380.42151)
  MoveL 8891 to (463.81, 520.3, 160) mm, rotated rx -180 ry 0 rz 160 deg; joints [9.517, 48.211, 10.273, -146.411, 62.942, 163.19]
  Call Extruder(383.15637)
  MoveL 8892 to (463.41, 519.57, 160) mm, rotated rx -180 ry 0 rz 160 deg; joints [9.428, 48.134, 10.42, -146.527, 62.975, 163.277]
  Call Extruder(385.87063)
  MoveL 8893 to (463.03, 518.84, 160) mm, rotated rx 180 ry 0 rz 160 deg; joints [9.337, 48.061, 10.561, -146.643, 63.006, 163.363]
  Call Extruder(388.80415)
  MoveL 8894 to (462.63, 518.04, 160) mm, rotated rx 180 ry 0 rz 160 deg; joints [9.238, 47.984, 10.71, -146.769, 63.037, 163.456]
  Set speed (17.1 mm/s)
  Call Extruder(394.40802)
  MoveL 8895 to (461.93, 516.5, 160) mm, rotated rx -180 ry 0 rz 160 deg; joints [9.044, 47.843, 10.98, -147.014, 63.091, 163.63]
  Call Extruder(399.78989)
  MoveL 8896 to (461.31, 514.98, 160) mm, rotated rx -180 ry 0 rz 160 deg; joints [8.851, 47.718, 11.22, -147.253, 63.134, 163.794]
  Set speed (17.1 mm/s)
  Call Extruder(401.63377)
  MoveL 8897 to (461.11, 514.46, 160) mm, rotated rx 180 ry 0 rz 160 deg; joints [8.784, 47.678, 11.299, -147.336, 63.147, 163.85]
  Set speed (17.1 mm/s)
  Call Extruder(405.43722)
  MoveL 8898 to (460.72, 513.38, 160) mm, rotated rx -180 ry 0 rz 160 deg; joints [8.644, 47.597, 11.454, -147.507, 63.171, 163.963]
  Set speed (17.1 mm/s)
  Call Extruder(410.94875)
  MoveL 8899 to (460.22, 511.78, 160) mm, rotated rx -180 ry 0 rz 160 deg; joints [8.437, 47.488, 11.664, -147.758, 63.199, 164.124]
  Set speed (17.1 mm/s)
  Call Extruder(413.97456)
  MoveL 8900 to (459.97, 510.9, 160) mm, rotated rx 180 ry 0 rz 160 deg; joints [8.321, 47.433, 11.77, -147.897, 63.211, 164.211]
  Set speed (17.1 mm/s)
  Call Extruder(416.61700)
  MoveL 8901 to (459.76, 510.12, 160) mm, rotated rx 180 ry 0 rz 160 deg; joints [8.219, 47.387, 11.859, -148.018, 63.219, 164.286]
  Set speed (17.1 mm/s)
  Call Extruder(418.99234)
  MoveL 8902 to (459.6, 509.42, 160) mm, rotated rx -180 ry 0 rz 160 deg; joints [8.126, 47.348, 11.934, -148.128, 63.225, 164.352]
  Set speed (17.1 mm/s)
  Call Extruder(422.53192)
  MoveL 8903 to (459.36, 508.38, 160) mm, rotated rx 180 ry 0 rz 160 deg; joints [7.987, 47.293, 12.041, -148.292, 63.231, 164.45]
  Set speed (17.1 mm/s)
  Call Extruder(428.00919)
  MoveL 8904 to (459.06, 506.74, 160) mm, rotated rx -180 ry 0 rz 160 deg; joints [7.767, 47.216, 12.189, -148.547, 63.233, 164.598]
  Call Extruder(433.60729)
  MoveL 8905 to (458.82, 505.06, 160) mm, rotated rx 180 ry 0 rz 160 deg; joints [7.54, 47.148, 12.319, -148.809, 63.227, 164.746]
  Set speed (17.1 mm/s)
  Call Extruder(439.19088)
  MoveL 8906 to (458.64, 503.38, 160) mm, rotated rx -180 ry 0 rz 160 deg; joints [7.311, 47.091, 12.429, -149.071, 63.212, 164.888]
  Set speed (17.1 mm/s)
  Call Extruder(444.80785)
  MoveL 8907 to (458.54, 501.68, 160) mm, rotated rx -180 ry 0 rz 160 deg; joints [7.077, 47.045, 12.518, -149.334, 63.188, 165.026]
  Set speed (17.1 mm/s)
  Call Extruder(450.24689)
  MoveL 8908 to (458.51, 500.03, 160) mm, rotated rx -180 ry 0 rz 160 deg; joints [6.849, 47.011, 12.583, -149.589, 63.156, 165.156]
  Set speed (17.1 mm/s)
  Call Extruder(455.16792)
  MoveL 8909 to (458.54, 498.53, 160) mm, rotated rx -180 ry 0 rz 160 deg; joints [6.642, 46.989, 12.625, -149.819, 63.121, 165.269]
  Set speed (17.1 mm/s)
  Call Extruder(460.35667)
  MoveL 8910 to (458.62, 496.96, 160) mm, rotated rx 180 ry 0 rz 160 deg; joints [6.423, 46.975, 12.652, -150.06, 63.076, 165.383]
  Set speed (17.1 mm/s)
  Call Extruder(465.23032)
  MoveL 8911 to (458.75, 495.49, 160) mm, rotated rx -180 ry 0 rz 160 deg; joints [6.217, 46.971, 12.66, -150.285, 63.028, 165.487]
  Set speed (17.1 mm/s)
  Call Extruder(470.42563)
  MoveL 8912 to (458.96, 493.93, 160) mm, rotated rx 180 ry 0 rz 160 deg; joints [5.997, 46.976, 12.651, -150.523, 62.969, 165.593]
  Set speed (17.1 mm/s)
  Call Extruder(475.54885)
  MoveL 8913 to (459.21, 492.39, 160) mm, rotated rx 180 ry 0 rz 160 deg; joints [5.78, 46.99, 12.623, -150.755, 62.904, 165.693]
  Set speed (17.1 mm/s)
  Call Extruder(480.41728)
  MoveL 8914 to (459.51, 490.94, 160) mm, rotated rx 180 ry 0 rz 160 deg; joints [5.575, 47.013, 12.58, -150.974, 62.835, 165.783]
  Call Extruder(485.68258)
  MoveL 8915 to (459.89, 489.39, 160) mm, rotated rx 180 ry 0 rz 160 deg; joints [5.355, 47.046, 12.516, -151.206, 62.754, 165.877]
  Set speed (17.1 mm/s)
  Call Extruder(490.55399)
  MoveL 8916 to (460.29, 487.97, 160) mm, rotated rx 180 ry 0 rz 160 deg; joints [5.152, 47.086, 12.439, -151.418, 62.672, 165.958]
  Call Extruder(495.51887)
  MoveL 8917 to (460.76, 486.54, 160) mm, rotated rx -180 ry 0 rz 160 deg; joints [4.948, 47.135, 12.345, -151.63, 62.583, 166.036]
  Set speed (17.1 mm/s)
  Call Extruder(500.53953)
  MoveL 8918 to (461.27, 485.11, 160) mm, rotated rx 180 ry 0 rz 160 deg; joints [4.743, 47.193, 12.233, -151.841, 62.487, 166.111]
  Set speed (17.1 mm/s)
  Call Extruder(505.75870)
  MoveL 8919 to (461.87, 483.64, 160) mm, rotated rx -180 ry 0 rz 160 deg; joints [4.533, 47.262, 12.099, -152.055, 62.379, 166.183]
  Call Extruder(510.74916)
  MoveL 8920 to (462.49, 482.26, 160) mm, rotated rx 180 ry 0 rz 160 deg; joints [4.335, 47.338, 11.954, -152.255, 62.271, 166.247]
  Set speed (17.1 mm/s)
  Call Extruder(515.69821)
  MoveL 8921 to (463.16, 480.92, 160) mm, rotated rx 180 ry 0 rz 160 deg; joints [4.143, 47.421, 11.794, -152.447, 62.157, 166.305]
  Set speed (17.1 mm/s)
  Call Extruder(520.77468)
  MoveL 8922 to (463.89, 479.56, 160) mm, rotated rx -180 ry 0 rz 160 deg; joints [3.949, 47.514, 11.614, -152.64, 62.034, 166.36]
  Set speed (17.1 mm/s)
  Call Extruder(525.85850)
  MoveL 8923 to (464.68, 478.24, 160) mm, rotated rx -180 ry 0 rz 160 deg; joints [3.758, 47.617, 11.417, -152.826, 61.905, 166.409]
  Set speed (17.1 mm/s)
  Call Extruder(530.84905)
  MoveL 8924 to (465.49, 476.96, 160) mm, rotated rx 180 ry 0 rz 160 deg; joints [3.575, 47.725, 11.208, -153.003, 61.773, 166.452]
  Set speed (17.1 mm/s)
  Call Extruder(535.87717)
  MoveL 8925 to (466.37, 475.71, 160) mm, rotated rx -180 ry 0 rz 160 deg; joints [3.396, 47.842, 10.982, -153.175, 61.634, 166.491]
  Set speed (17.1 mm/s)
  Call Extruder(540.74161)
  MoveL 8926 to (467.25, 474.52, 160) mm, rotated rx -180 ry 0 rz 160 deg; joints [3.227, 47.963, 10.749, -153.335, 61.494, 166.522]
  Set speed (17.1 mm/s)
  Call Extruder(545.89010)
  MoveL 8927 to (468.23, 473.31, 160) mm, rotated rx 180 ry 0 rz 160 deg; joints [3.053, 48.099, 10.488, -153.497, 61.342, 166.551]
  Set speed (17.1 mm/s)
  Call Extruder(551.18137)
  MoveL 8928 to (469.29, 472.1, 160) mm, rotated rx 180 ry 0 rz 160 deg; joints [2.88, 48.247, 10.203, -153.655, 61.179, 166.573]
  Set speed (17.1 mm/s)
  Call Extruder(555.94666)
  MoveL 8929 to (470.28, 471.05, 160) mm, rotated rx 180 ry 0 rz 160 deg; joints [2.73, 48.387, 9.933, -153.79, 61.028, 166.588]
  Call Extruder(561.05717)
  MoveL 8930 to (471.38, 469.96, 160) mm, rotated rx -180 ry 0 rz 160 deg; joints [2.575, 48.545, 9.63, -153.927, 60.861, 166.599]
  Set speed (17.1 mm/s)
  Call Extruder(566.02733)
  MoveL 8931 to (472.49, 468.94, 160) mm, rotated rx 180 ry 0 rz 160 deg; joints [2.43, 48.705, 9.322, -154.053, 60.694, 166.603]
  Set speed (17.1 mm/s)
  Call Extruder(571.20764)
  MoveL 8932 to (473.69, 467.92, 160) mm, rotated rx -180 ry 0 rz 160 deg; joints [2.285, 48.878, 8.988, -154.175, 60.516, 166.602]
  Set speed (17.1 mm/s)
  Call Extruder(576.39020)
  MoveL 8933 to (474.92, 466.95, 160) mm, rotated rx 180 ry 0 rz 160 deg; joints [2.147, 49.059, 8.639, -154.288, 60.334, 166.595]
  Set speed (17.1 mm/s)
  Call Extruder(581.06917)
  MoveL 8934 to (476.07, 466.11, 160) mm, rotated rx 180 ry 0 rz 160 deg; joints [2.028, 49.228, 8.314, -154.382, 60.165, 166.583]
  Set speed (17.1 mm/s)
  Call Extruder(586.15227)
  MoveL 8935 to (477.35, 465.24, 160) mm, rotated rx 180 ry 0 rz 160 deg; joints [1.906, 49.418, 7.949, -154.476, 59.979, 166.564]
  Set speed (17.1 mm/s)
  Call Extruder(591.33807)
  MoveL 8936 to (478.68, 464.41, 160) mm, rotated rx -180 ry 0 rz 160 deg; joints [1.789, 49.617, 7.565, -154.562, 59.785, 166.538]
  Set speed (17.1 mm/s)
  Call Extruder(596.37114)
  MoveL 8937 to (480, 463.65, 160) mm, rotated rx 180 ry 0 rz 160 deg; joints [1.682, 49.817, 7.182, -154.636, 59.594, 166.508]
  Set speed (17.1 mm/s)
  Call Extruder(601.42179)
  MoveL 8938 to (481.36, 462.93, 160) mm, rotated rx -180 ry 0 rz 160 deg; joints [1.581, 50.022, 6.787, -154.701, 59.399, 166.471]
  Call Extruder(606.25810)
  MoveL 8939 to (482.68, 462.3, 160) mm, rotated rx -180 ry 0 rz 160 deg; joints [1.492, 50.224, 6.399, -154.755, 59.209, 166.43]
  Set speed (17.1 mm/s)
  Call Extruder(611.48290)
  MoveL 8940 to (484.13, 461.66, 160) mm, rotated rx -180 ry 0 rz 160 deg; joints [1.403, 50.446, 5.97, -154.803, 59.002, 166.379]
  Call Extruder(616.36236)
  MoveL 8941 to (485.51, 461.12, 160) mm, rotated rx 180 ry 0 rz 160 deg; joints [1.328, 50.659, 5.561, -154.838, 58.807, 166.326]
  Set speed (17.1 mm/s)
  Call Extruder(621.56332)
  MoveL 8942 to (487, 460.6, 160) mm, rotated rx -180 ry 0 rz 160 deg; joints [1.255, 50.89, 5.117, -154.866, 58.596, 166.263]
  Set speed (17.1 mm/s)
  Call Extruder(626.42466)
  MoveL 8943 to (488.41, 460.16, 160) mm, rotated rx 180 ry 0 rz 160 deg; joints [1.194, 51.11, 4.694, -154.883, 58.398, 166.198]
  Set speed (17.1 mm/s)
  Call Extruder(631.38792)
  MoveL 8944 to (489.86, 459.77, 160) mm, rotated rx -180 ry 0 rz 160 deg; joints [1.138, 51.338, 4.256, -154.891, 58.194, 166.127]
  Set speed (17.1 mm/s)
  Call Extruder(636.66218)
  MoveL 8945 to (491.42, 459.41, 160) mm, rotated rx -180 ry 0 rz 160 deg; joints [1.087, 51.584, 3.782, -154.889, 57.976, 166.044]
  Set speed (17.1 mm/s)
  Call Extruder(641.54359)
  MoveL 8946 to (492.88, 459.13, 160) mm, rotated rx 180 ry 0 rz 160 deg; joints [1.047, 51.815, 3.338, -154.878, 57.774, 165.961]
  Set speed (17.1 mm/s)
  Call Extruder(646.68907)
  MoveL 8947 to (494.42, 458.89, 160) mm, rotated rx 180 ry 0 rz 160 deg; joints [1.013, 52.061, 2.865, -154.857, 57.56, 165.869]
  Set speed (17.1 mm/s)
  Call Extruder(651.55231)
  MoveL 8948 to (495.88, 458.71, 160) mm, rotated rx -180 ry 0 rz 160 deg; joints [0.987, 52.296, 2.413, -154.827, 57.357, 165.775]
  Call Extruder(656.64359)
  MoveL 8949 to (497.42, 458.59, 160) mm, rotated rx 180 ry 0 rz 160 deg; joints [0.968, 52.545, 1.935, -154.787, 57.145, 165.671]
  Set speed (17.1 mm/s)
  Call Extruder(661.83714)
  MoveL 8950 to (499, 458.52, 160) mm, rotated rx -180 ry 0 rz 160 deg; joints [0.956, 52.8, 1.444, -154.736, 56.928, 165.559]
  Set speed (17.1 mm/s)
  Call Extruder(666.78298)
  MoveL 8951 to (500.5, 458.51, 160) mm, rotated rx -180 ry 0 rz 160 deg; joints [0.951, 53.046, 0.972, -154.678, 56.723, 165.446]
  Set speed (17.1 mm/s)
  Call Extruder(671.88742)
  MoveL 8952 to (502.05, 458.56, 160) mm, rotated rx -180 ry 0 rz 160 deg; joints [0.954, 53.3, 0.483, -154.608, 56.512, 165.324]
  Set speed (17.1 mm/s)
  Call Extruder(676.87674)
  MoveL 8953 to (503.56, 458.66, 160) mm, rotated rx 180 ry 0 rz 160 deg; joints [0.964, 53.55, 0.003, -154.531, 56.306, 165.199]
  Set speed (17.1 mm/s)
  Call Extruder(681.97896)
  MoveL 8954 to (505.1, 458.82, 160) mm, rotated rx 180 ry 0 rz 160 deg; joints [0.981, 53.806, -0.489, -154.444, 56.098, 165.066]
  Set speed (17.1 mm/s)
  Call Extruder(686.86569)
  MoveL 8955 to (506.56, 459.03, 160) mm, rotated rx 180 ry 0 rz 160 deg; joints [1.004, 54.052, -0.961, -154.351, 55.9, 164.933]
  Set speed (17.1 mm/s)
  Call Extruder(691.81233)
  MoveL 8956 to (508.04, 459.3, 160) mm, rotated rx -180 ry 0 rz 160 deg; joints [1.034, 54.301, -1.439, -154.248, 55.701, 164.793]
  Call Extruder(696.28956)
  MoveL 8957 to (509.37, 459.58, 160) mm, rotated rx 180 ry 0 rz 160 deg; joints [1.066, 54.526, -1.871, -154.149, 55.523, 164.662]
  Call Extruder(701.94683)
  MoveL 8958 to (511.03, 460, 160) mm, rotated rx -180 ry 0 rz 160 deg; joints [1.115, 54.809, -2.416, -154.013, 55.301, 164.491]
  Set speed (17.1 mm/s)
  Call Extruder(707.07036)
  MoveL 8959 to (512.52, 460.44, 160) mm, rotated rx -180 ry 0 rz 160 deg; joints [1.166, 55.065, -2.908, -153.881, 55.103, 164.331]
  Set speed (17.1 mm/s)
  Call Extruder(712.00195)
  MoveL 8960 to (513.94, 460.92, 160) mm, rotated rx 180 ry 0 rz 160 deg; joints [1.222, 55.31, -3.378, -153.746, 54.916, 164.172]
  Set speed (17.1 mm/s)
  Call Extruder(717.11569)
  MoveL 8961 to (515.39, 461.47, 160) mm, rotated rx -180 ry 0 rz 160 deg; joints [1.286, 55.563, -3.863, -153.598, 54.725, 164.003]
  Set speed (17.1 mm/s)
  Call Extruder(722.25281)
  MoveL 8962 to (516.83, 462.08, 160) mm, rotated rx -180 ry 0 rz 160 deg; joints [1.356, 55.815, -4.347, -153.442, 54.537, 163.828]
  Call Extruder(727.04185)
  MoveL 8963 to (518.15, 462.69, 160) mm, rotated rx -180 ry 0 rz 160 deg; joints [1.427, 56.048, -4.794, -153.29, 54.366, 163.661]
  Set speed (17.1 mm/s)
  Call Extruder(732.14787)
  MoveL 8964 to (519.53, 463.39, 160) mm, rotated rx -180 ry 0 rz 160 deg; joints [1.509, 56.294, -5.265, -153.12, 54.187, 163.48]
  Call Extruder(737.33280)
  MoveL 8965 to (520.9, 464.16, 160) mm, rotated rx 180 ry 0 rz 160 deg; joints [1.598, 56.54, -5.738, -152.94, 54.011, 163.291]
  Set speed (17.1 mm/s)
  Call Extruder(742.28457)
  MoveL 8966 to (522.18, 464.94, 160) mm, rotated rx -180 ry 0 rz 160 deg; joints [1.688, 56.772, -6.183, -152.762, 53.847, 163.108]
  Set speed (17.1 mm/s)
  Call Extruder(747.41702)
  MoveL 8967 to (523.49, 465.8, 160) mm, rotated rx 180 ry 0 rz 160 deg; joints [1.788, 57.009, -6.638, -152.571, 53.683, 162.914]
  Set speed (17.1 mm/s)
  Call Extruder(752.29139)
  MoveL 8968 to (524.69, 466.66, 160) mm, rotated rx 180 ry 0 rz 160 deg; joints [1.887, 57.23, -7.062, -152.384, 53.532, 162.728]
  Set speed (17.1 mm/s)
  Call Extruder(757.44014)
  MoveL 8969 to (525.93, 467.61, 160) mm, rotated rx 180 ry 0 rz 160 deg; joints [1.996, 57.459, -7.502, -152.181, 53.379, 162.528]
  Set speed (17.1 mm/s)
  Call Extruder(762.42772)
  MoveL 8970 to (527.09, 468.57, 160) mm, rotated rx 180 ry 0 rz 160 deg; joints [2.108, 57.677, -7.919, -151.98, 53.235, 162.332]
  Set speed (17.1 mm/s)
  Call Extruder(767.39463)
  MoveL 8971 to (528.21, 469.58, 160) mm, rotated rx -180 ry 0 rz 160 deg; joints [2.223, 57.889, -8.326, -151.773, 53.099, 162.135]
  Call Extruder(772.62514)
  MoveL 8972 to (529.36, 470.68, 160) mm, rotated rx -180 ry 0 rz 160 deg; joints [2.35, 58.107, -8.744, -151.551, 52.962, 161.926]
  Set speed (17.1 mm/s)
  Call Extruder(775.51546)
  MoveL 8973 to (529.97, 471.31, 160) mm, rotated rx 180 ry 0 rz 160 deg; joints [2.421, 58.225, -8.97, -151.427, 52.889, 161.81]
  Set speed (17.1 mm/s)
  Call Extruder(778.24514)
  MoveL 8974 to (530.54, 471.91, 160) mm, rotated rx -180 ry 0 rz 160 deg; joints [2.49, 58.334, -9.18, -151.308, 52.823, 161.7]
  Set speed (17.1 mm/s)
  Call Extruder(780.90685)
  MoveL 8975 to (531.08, 472.51, 160) mm, rotated rx 180 ry 0 rz 160 deg; joints [2.559, 58.439, -9.381, -151.191, 52.76, 161.592]
  Set speed (17.1 mm/s)
  Call Extruder(783.86475)
  MoveL 8976 to (531.67, 473.19, 160) mm, rotated rx 180 ry 0 rz 160 deg; joints [2.637, 58.554, -9.602, -151.06, 52.692, 161.472]
  Set speed (17.1 mm/s)
  Call Extruder(786.51061)
  MoveL 8977 to (532.18, 473.81, 160) mm, rotated rx -180 ry 0 rz 160 deg; joints [2.707, 58.655, -9.795, -150.942, 52.634, 161.365]
  Call Extruder(789.25856)
  MoveL 8978 to (532.7, 474.46, 160) mm, rotated rx -180 ry 0 rz 160 deg; joints [2.782, 58.758, -9.992, -150.818, 52.575, 161.253]
  Set speed (17.1 mm/s)
  Call Extruder(794.37760)
  MoveL 8979 to (533.63, 475.7, 160) mm, rotated rx 180 ry 0 rz 160 deg; joints [2.923, 58.944, -10.35, -150.585, 52.472, 161.045]
  Call Extruder(797.68576)
  MoveL 8980 to (534.21, 476.52, 160) mm, rotated rx 180 ry 0 rz 160 deg; joints [3.016, 59.061, -10.574, -150.433, 52.409, 160.911]
  Set speed (17.1 mm/s)
  Call Extruder(800.48287)
  MoveL 8981 to (534.68, 477.23, 160) mm, rotated rx 180 ry 0 rz 160 deg; joints [3.097, 59.157, -10.758, -150.304, 52.359, 160.797]
  Call Extruder(803.27851)
  MoveL 8982 to (535.14, 477.94, 160) mm, rotated rx -180 ry 0 rz 160 deg; joints [3.178, 59.251, -10.938, -150.174, 52.311, 160.684]
  Set speed (17.1 mm/s)
  Call Extruder(805.99155)
  MoveL 8983 to (535.57, 478.64, 160) mm, rotated rx -180 ry 0 rz 160 deg; joints [3.258, 59.34, -11.109, -150.047, 52.266, 160.574]
  Set speed (17.1 mm/s)
  Call Extruder(808.88655)
  MoveL 8984 to (536.01, 479.4, 160) mm, rotated rx -180 ry 0 rz 160 deg; joints [3.344, 59.433, -11.287, -149.911, 52.221, 160.457]
  Set speed (17.1 mm/s)
  Call Extruder(813.32771)
  MoveL 8985 to (536.67, 480.57, 160) mm, rotated rx 180 ry 0 rz 160 deg; joints [3.478, 59.571, -11.55, -149.703, 52.157, 160.279]
  Set speed (17.1 mm/s)
  Call Extruder(817.26448)
  MoveL 8986 to (537.21, 481.64, 160) mm, rotated rx -180 ry 0 rz 160 deg; joints [3.599, 59.686, -11.772, -149.517, 52.107, 160.123]
  Set speed (17.1 mm/s)
  Call Extruder(822.07578)
  MoveL 8987 to (537.83, 482.96, 160) mm, rotated rx 180 ry 0 rz 160 deg; joints [3.749, 59.823, -12.034, -149.289, 52.05, 159.932]
  Set speed (17.1 mm/s)
  Call Extruder(828.49516)
  MoveL 8988 to (538.59, 484.76, 160) mm, rotated rx -180 ry 0 rz 160 deg; joints [3.953, 59.992, -12.357, -148.983, 51.988, 159.682]
  Set speed (17.1 mm/s)
  Call Extruder(834.20649)
  MoveL 8989 to (539.19, 486.38, 160) mm, rotated rx 180 ry 0 rz 160 deg; joints [4.138, 60.131, -12.624, -148.712, 51.944, 159.463]
  Call Extruder(839.59457)
  MoveL 8990 to (539.7, 487.93, 160) mm, rotated rx -180 ry 0 rz 160 deg; joints [4.315, 60.251, -12.855, -148.457, 51.912, 159.26]
  Call Extruder(845.11075)
  MoveL 8991 to (540.15, 489.55, 160) mm, rotated rx 180 ry 0 rz 160 deg; joints [4.498, 60.364, -13.07, -148.197, 51.89, 159.057]
  Set speed (17.1 mm/s)
  Call Extruder(850.69633)
  MoveL 8992 to (540.55, 491.19, 160) mm, rotated rx -180 ry 0 rz 160 deg; joints [4.686, 60.466, -13.266, -147.935, 51.877, 158.856]
  Call Extruder(856.40688)
  MoveL 8993 to (540.88, 492.89, 160) mm, rotated rx 180 ry 0 rz 160 deg; joints [4.88, 60.559, -13.444, -147.669, 51.876, 158.657]
  Set speed (17.1 mm/s)
  Call Extruder(862.00522)
  MoveL 8994 to (541.13, 494.57, 160) mm, rotated rx -180 ry 0 rz 160 deg; joints [5.072, 60.638, -13.595, -147.411, 51.885, 158.467]
  Call Extruder(867.69322)
  MoveL 8995 to (541.32, 496.29, 160) mm, rotated rx -180 ry 0 rz 160 deg; joints [5.269, 60.706, -13.725, -147.153, 51.905, 158.281]
  Set speed (17.1 mm/s)
  Call Extruder(873.20006)
  MoveL 8996 to (541.44, 497.95, 160) mm, rotated rx -180 ry 0 rz 160 deg; joints [5.461, 60.759, -13.827, -146.906, 51.936, 158.108]
  Set speed (17.1 mm/s)
  Call Extruder(878.78622)
  MoveL 8997 to (541.49, 499.65, 160) mm, rotated rx -180 ry 0 rz 160 deg; joints [5.656, 60.801, -13.907, -146.659, 51.977, 157.94]
  Set speed (17.1 mm/s)
  Call Extruder(884.24952)
  MoveL 8998 to (541.47, 501.3, 160) mm, rotated rx -180 ry 0 rz 160 deg; joints [5.848, 60.83, -13.963, -146.422, 52.027, 157.782]
  Set speed (17.1 mm/s)
  Call Extruder(889.95813)
  MoveL 8999 to (541.38, 503.04, 160) mm, rotated rx -180 ry 0 rz 160 deg; joints [6.049, 60.848, -13.998, -146.179, 52.089, 157.626]
  Set speed (17.1 mm/s)
  Call Extruder(895.46564)
  MoveL 9000 to (541.22, 504.7, 160) mm, rotated rx 180 ry 0 rz 160 deg; joints [6.243, 60.852, -14.006, -145.95, 52.16, 157.483]
  Set speed (17.1 mm/s)
  Call Extruder(901.24748)
  MoveL 9001 to (540.99, 506.44, 160) mm, rotated rx 180 ry 0 rz 160 deg; joints [6.446, 60.844, -13.99, -145.716, 52.245, 157.343]
  Call Extruder(906.74645)
  MoveL 9002 to (540.7, 508.08, 160) mm, rotated rx 180 ry 0 rz 160 deg; joints [6.64, 60.824, -13.952, -145.498, 52.334, 157.218]
  Set speed (17.1 mm/s)
  Call Extruder(912.38430)
  MoveL 9003 to (540.33, 509.75, 160) mm, rotated rx -180 ry 0 rz 160 deg; joints [6.838, 60.791, -13.888, -145.281, 52.436, 157.099]
  Set speed (17.1 mm/s)
  Call Extruder(917.82739)
  MoveL 9004 to (539.91, 511.35, 160) mm, rotated rx -180 ry 0 rz 160 deg; joints [7.028, 60.746, -13.803, -145.078, 52.544, 156.994]
  Set speed (17.1 mm/s)
  Call Extruder(923.55774)
  MoveL 9005 to (539.4, 513.01, 160) mm, rotated rx -180 ry 0 rz 160 deg; joints [7.227, 60.687, -13.689, -144.872, 52.666, 156.894]
  Set speed (17.1 mm/s)
  Call Extruder(929.29369)
  MoveL 9006 to (538.82, 514.65, 160) mm, rotated rx 180 ry 0 rz 160 deg; joints [7.425, 60.615, -13.551, -144.672, 52.798, 156.803]
  Set speed (17.1 mm/s)
  Call Extruder(934.81348)
  MoveL 9007 to (538.2, 516.21, 160) mm, rotated rx -180 ry 0 rz 160 deg; joints [7.614, 60.533, -13.395, -144.487, 52.933, 156.726]
  Set speed (17.1 mm/s)
  Call Extruder(940.25396)
  MoveL 9008 to (537.52, 517.72, 160) mm, rotated rx -180 ry 0 rz 160 deg; joints [7.799, 60.442, -13.22, -144.311, 53.075, 156.659]
  Call Extruder(943.15007)
  MoveL 9009 to (537.14, 518.51, 160) mm, rotated rx -180 ry 0 rz 160 deg; joints [7.896, 60.389, -13.118, -144.221, 53.153, 156.627]
  Set speed (17.1 mm/s)
  Call Extruder(945.94939)
  MoveL 9010 to (536.75, 519.26, 160) mm, rotated rx -180 ry 0 rz 160 deg; joints [7.99, 60.335, -13.014, -144.135, 53.23, 156.599]
  Set speed (17.1 mm/s)
  Call Extruder(948.64484)
  MoveL 9011 to (536.36, 519.98, 160) mm, rotated rx 180 ry 0 rz 160 deg; joints [8.08, 60.279, -12.908, -144.055, 53.307, 156.575]
  Set speed (17.1 mm/s)
  Call Extruder(951.55709)
  MoveL 9012 to (535.93, 520.75, 160) mm, rotated rx 180 ry 0 rz 160 deg; joints [8.176, 60.216, -12.788, -143.97, 53.392, 156.551]
  Call Extruder(954.32035)
  MoveL 9013 to (535.5, 521.47, 160) mm, rotated rx -180 ry 0 rz 160 deg; joints [8.266, 60.155, -12.669, -143.891, 53.474, 156.531]
  Call Extruder(957.15613)
  MoveL 9014 to (535.05, 522.21, 160) mm, rotated rx 180 ry 0 rz 160 deg; joints [8.359, 60.088, -12.542, -143.812, 53.559, 156.513]
  Set speed (17.1 mm/s)
  Call Extruder(959.89396)
  MoveL 9015 to (534.6, 522.9, 160) mm, rotated rx -180 ry 0 rz 160 deg; joints [8.447, 60.021, -12.414, -143.738, 53.644, 156.498]
  Set speed (17.1 mm/s)
  Call Extruder(962.84910)
  MoveL 9016 to (534.1, 523.64, 160) mm, rotated rx -180 ry 0 rz 160 deg; joints [8.542, 59.946, -12.27, -143.66, 53.737, 156.485]
  Set speed (17.1 mm/s)
  Call Extruder(965.49397)
  MoveL 9017 to (533.63, 524.3, 160) mm, rotated rx 180 ry 0 rz 160 deg; joints [8.626, 59.877, -12.137, -143.592, 53.822, 156.475]
  Set speed (17.1 mm/s)
  Call Extruder(968.34472)
  MoveL 9018 to (533.12, 525, 160) mm, rotated rx 180 ry 0 rz 160 deg; joints [8.716, 59.799, -11.987, -143.521, 53.915, 156.468]
  Call Extruder(971.08550)
  MoveL 9019 to (532.61, 525.66, 160) mm, rotated rx 180 ry 0 rz 160 deg; joints [8.801, 59.722, -11.84, -143.455, 54.006, 156.462]
  Set speed (17.1 mm/s)
  Call Extruder(973.87408)
  MoveL 9020 to (532.08, 526.31, 160) mm, rotated rx -180 ry 0 rz 160 deg; joints [8.887, 59.641, -11.685, -143.389, 54.1, 156.46]
  Set speed (17.1 mm/s)
  Call Extruder(978.31738)
  MoveL 9021 to (531.21, 527.35, 160) mm, rotated rx -180 ry 0 rz 160 deg; joints [9.023, 59.507, -11.429, -143.288, 54.253, 156.46]
  Set speed (17.1 mm/s)
  Call Extruder(982.30945)
  MoveL 9022 to (530.39, 528.24, 160) mm, rotated rx 180 ry 0 rz 160 deg; joints [9.143, 59.381, -11.187, -143.203, 54.393, 156.467]
  Set speed (17.1 mm/s)
  Call Extruder(985.12550)
  MoveL 9023 to (529.81, 528.86, 160) mm, rotated rx 180 ry 0 rz 160 deg; joints [9.226, 59.289, -11.011, -143.145, 54.494, 156.474]
  Set speed (17.1 mm/s)
  Call Extruder(987.86318)
  MoveL 9024 to (529.22, 529.46, 160) mm, rotated rx 180 ry 0 rz 160 deg; joints [9.306, 59.198, -10.836, -143.091, 54.593, 156.483]
  Set speed (17.1 mm/s)
  Call Extruder(990.64876)
  MoveL 9025 to (528.62, 530.04, 160) mm, rotated rx -180 ry 0 rz 160 deg; joints [9.387, 59.103, -10.654, -143.038, 54.694, 156.495]
  Set speed (17.1 mm/s)
  Call Extruder(993.46552)
  MoveL 9026 to (527.99, 530.63, 160) mm, rotated rx -180 ry 0 rz 160 deg; joints [9.467, 59.005, -10.466, -142.986, 54.798, 156.509]
  Set speed (17.1 mm/s)
  Call Extruder(998.55968)
  MoveL 9027 to (526.83, 531.65, 160) mm, rotated rx -180 ry 0 rz 160 deg; joints [9.609, 58.822, -10.115, -142.897, 54.989, 156.541]
  Set speed (17.1 mm/s)
  Call Extruder(1001.83011)
  MoveL 9028 to (526.07, 532.28, 160) mm, rotated rx -180 ry 0 rz 160 deg; joints [9.698, 58.7, -9.882, -142.845, 55.113, 156.566]
  Set speed (17.1 mm/s)
  Call Extruder(1006.14675)
  MoveL 9029 to (525.04, 533.09, 160) mm, rotated rx 180 ry 0 rz 160 deg; joints [9.814, 58.537, -9.568, -142.779, 55.278, 156.603]
  Set speed (17.1 mm/s)
  Call Extruder(1010.37856)
  MoveL 9030 to (524, 533.85, 160) mm, rotated rx -180 ry 0 rz 160 deg; joints [9.924, 58.371, -9.251, -142.72, 55.443, 156.645]
  Set speed (17.1 mm/s)
  Call Extruder(1013.05713)
  MoveL 9031 to (523.33, 534.31, 160) mm, rotated rx -180 ry 0 rz 160 deg; joints [9.992, 58.264, -9.046, -142.685, 55.548, 156.674]
  Set speed (17.1 mm/s)
  Call Extruder(1015.84196)
  MoveL 9032 to (522.63, 534.78, 160) mm, rotated rx -180 ry 0 rz 160 deg; joints [10.061, 58.152, -8.83, -142.65, 55.658, 156.706]
  Set speed (17.1 mm/s)
  Call Extruder(1019.08416)
  MoveL 9033 to (521.8, 535.3, 160) mm, rotated rx 180 ry 0 rz 160 deg; joints [10.141, 58.018, -8.573, -142.613, 55.787, 156.747]
  Set speed (17.1 mm/s)
  Call Extruder(1021.42665)
  MoveL 9034 to (521.19, 535.67, 160) mm, rotated rx -180 ry 0 rz 160 deg; joints [10.197, 57.92, -8.385, -142.587, 55.881, 156.778]
  Set speed (17.1 mm/s)
  Call Extruder(1026.42670)
  MoveL 9035 to (519.88, 536.42, 160) mm, rotated rx -180 ry 0 rz 160 deg; joints [10.314, 57.708, -7.979, -142.537, 56.081, 156.848]
  Set speed (17.1 mm/s)
  Call Extruder(1031.42504)
  MoveL 9036 to (518.54, 537.13, 160) mm, rotated rx 180 ry 0 rz 160 deg; joints [10.426, 57.491, -7.563, -142.494, 56.283, 156.925]
  Set speed (17.1 mm/s)
  Call Extruder(1035.37783)
  MoveL 9037 to (517.46, 537.64, 160) mm, rotated rx 180 ry 0 rz 160 deg; joints [10.511, 57.316, -7.227, -142.465, 56.444, 156.99]
  Set speed (17.1 mm/s)
  Call Extruder(1041.08907)
  MoveL 9038 to (515.87, 538.34, 160) mm, rotated rx 180 ry 0 rz 160 deg; joints [10.629, 57.058, -6.732, -142.43, 56.678, 157.092]
  Set speed (17.1 mm/s)
  Call Extruder(1046.45109)
  MoveL 9039 to (514.35, 538.93, 160) mm, rotated rx 180 ry 0 rz 160 deg; joints [10.733, 56.811, -6.258, -142.406, 56.898, 157.194]
  Set speed (17.1 mm/s)
  Call Extruder(1052.09899)
  MoveL 9040 to (512.74, 539.49, 160) mm, rotated rx -180 ry 0 rz 160 deg; joints [10.837, 56.547, -5.751, -142.388, 57.13, 157.309]
  Set speed (17.1 mm/s)
  Call Extruder(1054.99771)
  MoveL 9041 to (511.9, 539.75, 160) mm, rotated rx 180 ry 0 rz 160 deg; joints [10.887, 56.41, -5.488, -142.383, 57.25, 157.37]
  Set speed (17.1 mm/s)
  Call Extruder(1057.66030)
  MoveL 9042 to (511.12, 539.97, 160) mm, rotated rx -180 ry 0 rz 160 deg; joints [10.932, 56.283, -5.245, -142.379, 57.359, 157.428]
  Set speed (17.1 mm/s)
  Call Extruder(1060.09928)
